LIN {X 0,Y 368.671,Z 450.598,A -85,B 0,C 180,E1 -13029.655,E2 -13029.655} C_VEL
LIN {X 0,Y 367.52,Z 522.522,A -85,B 0,C 180,E1 -13031.066,E2 -13031.066} C_VEL
LIN {X 0,Y 366.94,Z 535.872,A -85,B 0,C 180,E1 -13031.542,E2 -13031.542} C_VEL
LIN {X 0,Y 366.16,Z 548.093,A -85,B 0,C 180,E1 -13032.188,E2 -13032.188} C_VEL
LIN {X 0,Y 365.203,Z 560.412,A -85,B 0,C 180,E1 -13033.079,E2 -13033.079} C_VEL
LIN {X 0,Y 364.125,Z 572.06,A -85,B 0,C 180,E1 -13034.18,E2 -13034.18} C_VEL
LIN {X 0,Y 363.279,Z 582.567,A -85,B 0,C 180,E1 -13035.434,E2 -13035.434} C_VEL
LIN {X 0,Y 362.416,Z 591.99,A -85,B 0,C 180,E1 -13036.829,E2 -13036.829} C_VEL
LIN {X 0,Y 361.757,Z 599.735,A -85,B 0,C 180,E1 -13038.23,E2 -13038.23} C_VEL
LIN {X 0,Y 361.125,Z 607.312,A -85,B 0,C 180,E1 -13039.913,E2 -13039.913} C_VEL
LIN {X 0,Y 360.708,Z 613.396,A -85,B 0,C 180,E1 -13041.598,E2 -13041.598} C_VEL
LIN {X 0,Y 360.485,Z 618.204,A -85,B 0,C 180,E1 -13043.283,E2 -13043.283} C_VEL
LIN {X 0,Y 360.41,Z 621.877,A -85,B 0,C 180,E1 -13044.966,E2 -13044.966} C_VEL
LIN {X 0,Y 360.355,Z 624.517,A -85,B 0,C 180,E1 -13046.646,E2 -13046.646} C_VEL
LIN {X 0,Y 360.397,Z 625.759,A -85,B 0,C 180,E1 -13047.765,E2 -13047.765} C_VEL
LIN {X 0,Y 360.475,Z 626.58,A -85,B 0,C 180,E1 -13048.883,E2 -13048.883} C_VEL
LIN {X 0,Y 360.477,Z 626.968,A -85,B 0,C 180,E1 -13050,E2 -13050} C_VEL
LIN {X 0,Y 360.453,Z 626.966,A -85,B 0,C 180,E1 -13051.117,E2 -13051.117} C_VEL
LIN {X 0,Y 360.353,Z 626.574,A -85,B 0,C 180,E1 -13052.235,E2 -13052.235} C_VEL
LIN {X 0,Y 360.326,Z 625.784,A -85,B 0,C 180,E1 -13053.354,E2 -13053.354} C_VEL
LIN {X 0,Y 360.371,Z 624.558,A -85,B 0,C 180,E1 -13054.474,E2 -13054.474} C_VEL
LIN {X 0,Y 360.378,Z 622.329,A -85,B 0,C 180,E1 -13055.962,E2 -13055.962} C_VEL
LIN {X 0,Y 360.659,Z 618.37,A -85,B 0,C 180,E1 -13057.84,E2 -13057.84} C_VEL
LIN {X 0,Y 361.044,Z 613.682,A -85,B 0,C 180,E1 -13059.524,E2 -13059.524} C_VEL
LIN {X 0,Y 361.799,Z 606.644,A -85,B 0,C 180,E1 -13061.485,E2 -13061.485} C_VEL
LIN {X 0,Y 362.838,Z 599.055,A -85,B 0,C 180,E1 -13063.155,E2 -13063.155} C_VEL
LIN {X 0,Y 363.751,Z 591.32,A -85,B 0,C 180,E1 -13064.547,E2 -13064.547} C_VEL
LIN {X 0,Y 364.891,Z 581.912,A -85,B 0,C 180,E1 -13065.93,E2 -13065.93} C_VEL
LIN {X 0,Y 366.159,Z 571.498,A -85,B 0,C 180,E1 -13067.163,E2 -13067.163} C_VEL
LIN {X 0,Y 367.506,Z 559.948,A -85,B 0,C 180,E1 -13068.249,E2 -13068.249} C_VEL
LIN {X 0,Y 368.692,Z 547.75,A -85,B 0,C 180,E1 -13069.124,E2 -13069.124} C_VEL
LIN {X 0,Y 369.773,Z 534.193,A -85,B 0,C 180,E1 -13069.824,E2 -13069.824} C_VEL
LIN {X 0,Y 370.417,Z 521.877,A -85,B 0,C 180,E1 -13070.248,E2 -13070.248} C_VEL
LIN {X 0,Y 371.759,Z 449.686,A -85,B 0,C 180,E1 -13071.68,E2 -13071.68} C_VEL
LIN {X 0,Y 368.14,Z 427.447,A -85,B 0,C 180,E1 -13072.406,E2 -13072.406} C_VEL
LIN {X 0,Y 365.405,Z 413.474,A -85,B 0,C 180,E1 -13072.911,E2 -13072.911} C_VEL
LIN {X 0,Y 366.879,Z 400.729,A -85,B 0,C 180,E1 -13075.797,E2 -13075.797} C_VEL
LIN {X 0,Y 366.457,Z 396.694,A -85,B 0,C 180,E1 -13076.787,E2 -13076.787} C_VEL
LIN {X 0,Y 364.259,Z 386.406,A -85,B 0,C 180,E1 -13079.468,E2 -13079.468} C_VEL
LIN {X 0,Y 361.866,Z 376.41,A -85,B 0,C 180,E1 -13082.24,E2 -13082.24} C_VEL
LIN {X 0,Y 361.866,Z 376.411,A -85,B 0,C 180,E1 -13085.636,E2 -13085.636} C_VEL
LIN {X 0,Y 361.868,Z 376.407,A -85,B 0,C 180,E1 -13089.026,E2 -13089.026} C_VEL
LIN {X 0,Y 361.834,Z 376.409,A -85,B 0,C 180,E1 -13092.828,E2 -13092.828} C_VEL
LIN {X 0,Y 361.908,Z 376.401,A -85,B 0,C 180,E1 -13095.931,E2 -13095.931} C_VEL
LIN {X 0,Y 361.902,Z 376.401,A -85,B 0,C 180,E1 -13099.231,E2 -13099.231} C_VEL
LIN {X 0,Y 361.864,Z 376.405,A -85,B 0,C 180,E1 -13102.982,E2 -13102.982} C_VEL
LIN {X 0,Y 361.853,Z 376.408,A -85,B 0,C 180,E1 -13106.63,E2 -13106.63} C_VEL
LIN {X 0,Y 361.87,Z 376.406,A -85,B 0,C 180,E1 -13109.672,E2 -13109.672} C_VEL
LIN {X 0,Y 361.948,Z 376.387,A -85,B 0,C 180,E1 -13113.475,E2 -13113.475} C_VEL
LIN {X 0,Y 361.883,Z 376.399,A -85,B 0,C 180,E1 -13117.144,E2 -13117.144} C_VEL
LIN {X 0,Y 361.913,Z 376.398,A -85,B 0,C 180,E1 -13120.724,E2 -13120.724} C_VEL
LIN {X 0,Y 361.938,Z 376.395,A -85,B 0,C 180,E1 -13124.226,E2 -13124.226} C_VEL
LIN {X 0,Y 361.992,Z 376.391,A -85,B 0,C 180,E1 -13126.528,E2 -13126.528} C_VEL
LIN {X 0,Y 362.029,Z 376.382,A -85,B 0,C 180,E1 -13129.938,E2 -13129.938} C_VEL
LIN {X 0,Y 362.143,Z 376.373,A -85,B 0,C 180,E1 -13132.193,E2 -13132.193} C_VEL
LIN {X 0,Y 362.111,Z 376.37,A -85,B 0,C 180,E1 -13134.431,E2 -13134.431} C_VEL
LIN {X 0,Y 362.276,Z 376.353,A -85,B 0,C 180,E1 -13137.777,E2 -13137.777} C_VEL
LIN {X 0,Y 362.422,Z 376.336,A -85,B 0,C 180,E1 -13140,E2 -13140} C_VEL
LIN {X 0,Y 362.275,Z 376.357,A -85,B 0,C 180,E1 -13142.224,E2 -13142.224} C_VEL
LIN {X 0,Y 362.157,Z 376.373,A -85,B 0,C 180,E1 -13146.687,E2 -13146.687} C_VEL
LIN {X 0,Y 362.024,Z 376.388,A -85,B 0,C 180,E1 -13150.063,E2 -13150.063} C_VEL
LIN {X 0,Y 361.991,Z 376.39,A -85,B 0,C 180,E1 -13153.899,E2 -13153.899} C_VEL
LIN {X 0,Y 361.961,Z 376.393,A -85,B 0,C 180,E1 -13157.939,E2 -13157.939} C_VEL
LIN {X 0,Y 361.886,Z 376.402,A -85,B 0,C 180,E1 -13161.654,E2 -13161.654} C_VEL
LIN {X 0,Y 361.923,Z 376.39,A -85,B 0,C 180,E1 -13165.291,E2 -13165.291} C_VEL
LIN {X 0,Y 361.913,Z 376.391,A -85,B 0,C 180,E1 -13167.779,E2 -13167.779} C_VEL
LIN {X 0,Y 361.842,Z 376.407,A -85,B 0,C 180,E1 -13171.286,E2 -13171.286} C_VEL
LIN {X 0,Y 361.85,Z 376.411,A -85,B 0,C 180,E1 -13174.281,E2 -13174.281} C_VEL
LIN {X 0,Y 361.862,Z 376.408,A -85,B 0,C 180,E1 -13177.224,E2 -13177.224} C_VEL
LIN {X 0,Y 361.903,Z 376.407,A -85,B 0,C 180,E1 -13180.769,E2 -13180.769} C_VEL
LIN {X 0,Y 361.909,Z 376.411,A -85,B 0,C 180,E1 -13184.355,E2 -13184.355} C_VEL
LIN {X 0,Y 361.857,Z 376.415,A -85,B 0,C 180,E1 -13187.565,E2 -13187.565} C_VEL
LIN {X 0,Y 361.875,Z 376.41,A -85,B 0,C 180,E1 -13190.973,E2 -13190.973} C_VEL
LIN {X 0,Y 361.875,Z 376.41,A -85,B 0,C 180,E1 -13194.656,E2 -13194.656} C_VEL
LIN {X 0,Y 361.934,Z 376.564,A -85,B 0,C 180,E1 -13195.729,E2 -13195.729} C_VEL
LIN {X 0,Y 363.517,Z 383.858,A -85,B 0,C 180,E1 -13198.004,E2 -13198.004} C_VEL
LIN {X 0,Y 370.823,Z 401.263,A -85,B 0,C 180,E1 -13198.929,E2 -13198.929} C_VEL
LIN {X 0,Y 372.558,Z 408.259,A -85,B 0,C 180,E1 -13199.203,E2 -13199.203} C_VEL
LIN {X 0,Y 370.891,Z 490.155,A -85,B 0,C 180,E1 -13200.824,E2 -13200.824} C_VEL
LIN {X 0,Y 370.371,Z 502.076,A -85,B 0,C 180,E1 -13201.247,E2 -13201.247} C_VEL
LIN {X 0,Y 369.552,Z 514.899,A -85,B 0,C 180,E1 -13201.922,E2 -13201.922} C_VEL
LIN {X 0,Y 368.697,Z 524.869,A -85,B 0,C 180,E1 -13202.622,E2 -13202.622} C_VEL
LIN {X 0,Y 367.786,Z 535.953,A -85,B 0,C 180,E1 -13203.623,E2 -13203.623} C_VEL
LIN {X 0,Y 366.561,Z 546.433,A -85,B 0,C 180,E1 -13204.805,E2 -13204.805} C_VEL
LIN {X 0,Y 365.343,Z 556.155,A -85,B 0,C 180,E1 -13206.174,E2 -13206.174} C_VEL
LIN {X 0,Y 364.217,Z 564.926,A -85,B 0,C 180,E1 -13207.702,E2 -13207.702} C_VEL
LIN {X 0,Y 363.166,Z 572.436,A -85,B 0,C 180,E1 -13209.319,E2 -13209.319} C_VEL
LIN {X 0,Y 362.381,Z 577.833,A -85,B 0,C 180,E1 -13210.75,E2 -13210.75} C_VEL
LIN {X 0,Y 361.675,Z 583.349,A -85,B 0,C 180,E1 -13212.581,E2 -13212.581} C_VEL
LIN {X 0,Y 361.165,Z 587.097,A -85,B 0,C 180,E1 -13214.192,E2 -13214.192} C_VEL
LIN {X 0,Y 360.907,Z 589.153,A -85,B 0,C 180,E1 -13215.336,E2 -13215.336} C_VEL
LIN {X 0,Y 360.684,Z 591.358,A -85,B 0,C 180,E1 -13216.975,E2 -13216.975} C_VEL
LIN {X 0,Y 360.421,Z 592.768,A -85,B 0,C 180,E1 -13218.756,E2 -13218.756} C_VEL
LIN {X 0,Y 360.326,Z 593.102,A -85,B 0,C 180,E1 -13221.023,E2 -13221.023} C_VEL
LIN {X 0,Y 360.391,Z 592.689,A -85,B 0,C 180,E1 -13222.154,E2 -13222.154} C_VEL
LIN {X 0,Y 360.52,Z 591.294,A -85,B 0,C 180,E1 -13223.83,E2 -13223.83} C_VEL
LIN {X 0,Y 360.617,Z 587.969,A -85,B 0,C 180,E1 -13226.089,E2 -13226.089} C_VEL
LIN {X 0,Y 360.94,Z 584.326,A -85,B 0,C 180,E1 -13227.768,E2 -13227.768} C_VEL
LIN {X 0,Y 361.199,Z 579.599,A -85,B 0,C 180,E1 -13229.443,E2 -13229.443} C_VEL
LIN {X 0,Y 361.97,Z 572.495,A -85,B 0,C 180,E1 -13231.391,E2 -13231.391} C_VEL
LIN {X 0,Y 362.707,Z 564.761,A -85,B 0,C 180,E1 -13233.054,E2 -13233.054} C_VEL
LIN {X 0,Y 363.587,Z 555.113,A -85,B 0,C 180,E1 -13234.712,E2 -13234.712} C_VEL
LIN {X 0,Y 364.548,Z 545.11,A -85,B 0,C 180,E1 -13236.087,E2 -13236.087} C_VEL
LIN {X 0,Y 365.502,Z 533.787,A -85,B 0,C 180,E1 -13237.319,E2 -13237.319} C_VEL
LIN {X 0,Y 366.31,Z 522.692,A -85,B 0,C 180,E1 -13238.273,E2 -13238.273} C_VEL
LIN {X 0,Y 366.903,Z 511.497,A -85,B 0,C 180,E1 -13239.023,E2 -13239.023} C_VEL
LIN {X 0,Y 367.47,Z 498.848,A -85,B 0,C 180,E1 -13239.633,E2 -13239.633} C_VEL
LIN {X 0,Y 367.834,Z 485.603,A -85,B 0,C 180,E1 -13240.039,E2 -13240.039} C_VEL
LIN {X 0,Y 369.128,Z 406.287,A -85,B 0,C 180,E1 -13241.575,E2 -13241.575} C_VEL
LIN {X 0,Y 367.573,Z 397.862,A -85,B 0,C 180,E1 -13241.824,E2 -13241.824} C_VEL
LIN {X 0,Y 366.097,Z 394.053,A -85,B 0,C 180,E1 -13241.983,E2 -13241.983} C_VEL
LIN {X 0,Y 363.787,Z 390.703,A -85,B 0,C 180,E1 -13242.176,E2 -13242.176} C_VEL
LIN {X 0,Y 357.343,Z 384.3,A -85,B 0,C 180,E1 -13242.689,E2 -13242.689} C_VEL
LIN {X 0,Y 355.96,Z 382.402,A -85,B 0,C 180,E1 -13243.038,E2 -13243.038} C_VEL
LIN {X 0,Y 355.86,Z 382.081,A -85,B 0,C 180,E1 -13243.125,E2 -13243.125} C_VEL
LIN {X 0,Y 354.939,Z 377.274,A -85,B 0,C 180,E1 -13244.616,E2 -13244.616} C_VEL
LIN {X 0,Y 354.911,Z 377.279,A -85,B 0,C 180,E1 -13248.471,E2 -13248.471} C_VEL
LIN {X 0,Y 354.839,Z 377.284,A -85,B 0,C 180,E1 -13252.105,E2 -13252.105} C_VEL
LIN {X 0,Y 354.902,Z 377.274,A -85,B 0,C 180,E1 -13255.827,E2 -13255.827} C_VEL
LIN {X 0,Y 354.856,Z 377.279,A -85,B 0,C 180,E1 -13259.678,E2 -13259.678} C_VEL
LIN {X 0,Y 354.807,Z 377.286,A -85,B 0,C 180,E1 -13263.701,E2 -13263.701} C_VEL
LIN {X 0,Y 354.8,Z 377.292,A -85,B 0,C 180,E1 -13266.458,E2 -13266.458} C_VEL
LIN {X 0,Y 354.824,Z 377.283,A -85,B 0,C 180,E1 -13269.423,E2 -13269.423} C_VEL
LIN {X 0,Y 354.789,Z 377.289,A -85,B 0,C 180,E1 -13272.867,E2 -13272.867} C_VEL
LIN {X 0,Y 354.851,Z 377.284,A -85,B 0,C 180,E1 -13276.116,E2 -13276.116} C_VEL
LIN {X 0,Y 354.854,Z 377.279,A -85,B 0,C 180,E1 -13279.188,E2 -13279.188} C_VEL
LIN {X 0,Y 354.81,Z 377.29,A -85,B 0,C 180,E1 -13282.4,E2 -13282.4} C_VEL
LIN {X 0,Y 354.808,Z 377.286,A -85,B 0,C 180,E1 -13284.94,E2 -13284.94} C_VEL
LIN {X 0,Y 354.789,Z 377.292,A -85,B 0,C 180,E1 -13288.404,E2 -13288.404} C_VEL
LIN {X 0,Y 354.841,Z 377.282,A -85,B 0,C 180,E1 -13291.618,E2 -13291.618} C_VEL
LIN {X 0,Y 354.894,Z 377.28,A -85,B 0,C 180,E1 -13294.172,E2 -13294.172} C_VEL
LIN {X 0,Y 354.835,Z 377.285,A -85,B 0,C 180,E1 -13297.894,E2 -13297.894} C_VEL
LIN {X 0,Y 354.917,Z 377.275,A -85,B 0,C 180,E1 -13301.89,E2 -13301.89} C_VEL
LIN {X 0,Y 354.936,Z 377.273,A -85,B 0,C 180,E1 -13305.98,E2 -13305.98} C_VEL
LIN {X 0,Y 354.976,Z 377.266,A -85,B 0,C 180,E1 -13309.735,E2 -13309.735} C_VEL
LIN {X 0,Y 355.107,Z 377.253,A -85,B 0,C 180,E1 -13312.036,E2 -13312.036} C_VEL
LIN {X 0,Y 355.085,Z 377.255,A -85,B 0,C 180,E1 -13314.32,E2 -13314.32} C_VEL
LIN {X 0,Y 355.239,Z 377.234,A -85,B 0,C 180,E1 -13317.732,E2 -13317.732} C_VEL
LIN {X 0,Y 355.391,Z 377.218,A -85,B 0,C 180,E1 -13320,E2 -13320} C_VEL
LIN {X 0,Y 355.239,Z 377.236,A -85,B 0,C 180,E1 -13322.267,E2 -13322.267} C_VEL
LIN {X 0,Y 355.13,Z 377.245,A -85,B 0,C 180,E1 -13326.819,E2 -13326.819} C_VEL
LIN {X 0,Y 355.009,Z 377.26,A -85,B 0,C 180,E1 -13329.112,E2 -13329.112} C_VEL
LIN {X 0,Y 354.919,Z 377.273,A -85,B 0,C 180,E1 -13332.581,E2 -13332.581} C_VEL
LIN {X 0,Y 354.883,Z 377.282,A -85,B 0,C 180,E1 -13336.096,E2 -13336.096} C_VEL
LIN {X 0,Y 354.901,Z 377.275,A -85,B 0,C 180,E1 -13338.472,E2 -13338.472} C_VEL
LIN {X 0,Y 354.834,Z 377.287,A -85,B 0,C 180,E1 -13342.106,E2 -13342.106} C_VEL
LIN {X 0,Y 354.892,Z 377.279,A -85,B 0,C 180,E1 -13345.828,E2 -13345.828} C_VEL
LIN {X 0,Y 354.811,Z 377.288,A -85,B 0,C 180,E1 -13349.682,E2 -13349.682} C_VEL
LIN {X 0,Y 354.8,Z 377.29,A -85,B 0,C 180,E1 -13353.703,E2 -13353.703} C_VEL
LIN {X 0,Y 354.794,Z 377.288,A -85,B 0,C 180,E1 -13356.46,E2 -13356.46} C_VEL
LIN {X 0,Y 354.819,Z 377.285,A -85,B 0,C 180,E1 -13359.424,E2 -13359.424} C_VEL
LIN {X 0,Y 354.831,Z 377.282,A -85,B 0,C 180,E1 -13362.876,E2 -13362.876} C_VEL
LIN {X 0,Y 354.793,Z 377.291,A -85,B 0,C 180,E1 -13366.109,E2 -13366.109} C_VEL
LIN {X 0,Y 354.784,Z 377.289,A -85,B 0,C 180,E1 -13369.18,E2 -13369.18} C_VEL
LIN {X 0,Y 354.805,Z 377.287,A -85,B 0,C 180,E1 -13372.403,E2 -13372.403} C_VEL
LIN {X 0,Y 354.81,Z 377.285,A -85,B 0,C 180,E1 -13374.942,E2 -13374.942} C_VEL
LIN {X 0,Y 354.815,Z 377.285,A -85,B 0,C 180,E1 -13378.4,E2 -13378.4} C_VEL
LIN {X 0,Y 354.915,Z 377.465,A -85,B 0,C 180,E1 -13379.755,E2 -13379.755} C_VEL
LIN {X 0,Y 357.366,Z 389.378,A -85,B 0,C 180,E1 -13382.743,E2 -13382.743} C_VEL
LIN {X 0,Y 358.518,Z 396.453,A -85,B 0,C 180,E1 -13384.453,E2 -13384.453} C_VEL
LIN {X 0,Y 357.181,Z 410.658,A -85,B 0,C 180,E1 -13387.636,E2 -13387.636} C_VEL
LIN {X 0,Y 356.914,Z 413.639,A -85,B 0,C 180,E1 -13388.301,E2 -13388.301} C_VEL
LIN {X 0,Y 361.882,Z 450.204,A -85,B 0,C 180,E1 -13389.317,E2 -13389.317} C_VEL
LIN {X 0,Y 360.697,Z 522.605,A -85,B 0,C 180,E1 -13390.768,E2 -13390.768} C_VEL
LIN {X 0,Y 360.091,Z 535.816,A -85,B 0,C 180,E1 -13391.251,E2 -13391.251} C_VEL
LIN {X 0,Y 359.286,Z 547.966,A -85,B 0,C 180,E1 -13391.909,E2 -13391.909} C_VEL
LIN {X 0,Y 358.41,Z 559.427,A -85,B 0,C 180,E1 -13392.748,E2 -13392.748} C_VEL
LIN {X 0,Y 357.294,Z 571.201,A -85,B 0,C 180,E1 -13393.869,E2 -13393.869} C_VEL
LIN {X 0,Y 356.305,Z 581.79,A -85,B 0,C 180,E1 -13395.143,E2 -13395.143} C_VEL
LIN {X 0,Y 355.46,Z 591.324,A -85,B 0,C 180,E1 -13396.567,E2 -13396.567} C_VEL
LIN {X 0,Y 354.766,Z 599.127,A -85,B 0,C 180,E1 -13397.995,E2 -13397.995} C_VEL
LIN {X 0,Y 354.077,Z 606.751,A -85,B 0,C 180,E1 -13399.71,E2 -13399.71} C_VEL
LIN {X 0,Y 353.652,Z 612.881,A -85,B 0,C 180,E1 -13401.429,E2 -13401.429} C_VEL
LIN {X 0,Y 353.396,Z 617.727,A -85,B 0,C 180,E1 -13403.147,E2 -13403.147} C_VEL
LIN {X 0,Y 353.31,Z 621.436,A -85,B 0,C 180,E1 -13404.865,E2 -13404.865} C_VEL
LIN {X 0,Y 353.274,Z 624.111,A -85,B 0,C 180,E1 -13406.579,E2 -13406.579} C_VEL
LIN {X 0,Y 353.3,Z 625.37,A -85,B 0,C 180,E1 -13407.72,E2 -13407.72} C_VEL
LIN {X 0,Y 353.393,Z 626.221,A -85,B 0,C 180,E1 -13408.86,E2 -13408.86} C_VEL
LIN {X 0,Y 353.395,Z 626.626,A -85,B 0,C 180,E1 -13410,E2 -13410} C_VEL
LIN {X 0,Y 353.355,Z 626.639,A -85,B 0,C 180,E1 -13411.14,E2 -13411.14} C_VEL
LIN {X 0,Y 353.245,Z 625.498,A -85,B 0,C 180,E1 -13413.422,E2 -13413.422} C_VEL
LIN {X 0,Y 353.282,Z 624.294,A -85,B 0,C 180,E1 -13414.564,E2 -13414.564} C_VEL
LIN {X 0,Y 353.414,Z 620.653,A -85,B 0,C 180,E1 -13416.852,E2 -13416.852} C_VEL
LIN {X 0,Y 353.718,Z 616.737,A -85,B 0,C 180,E1 -13418.57,E2 -13418.57} C_VEL
LIN {X 0,Y 354.223,Z 611.706,A -85,B 0,C 180,E1 -13420.286,E2 -13420.286} C_VEL
LIN {X 0,Y 354.96,Z 605.411,A -85,B 0,C 180,E1 -13421.999,E2 -13421.999} C_VEL
LIN {X 0,Y 356.115,Z 597.563,A -85,B 0,C 180,E1 -13423.699,E2 -13423.699} C_VEL
LIN {X 0,Y 357.115,Z 589.198,A -85,B 0,C 180,E1 -13425.178,E2 -13425.178} C_VEL
LIN {X 0,Y 358.438,Z 578.813,A -85,B 0,C 180,E1 -13426.663,E2 -13426.663} C_VEL
LIN {X 0,Y 359.918,Z 567.735,A -85,B 0,C 180,E1 -13427.911,E2 -13427.911} C_VEL
LIN {X 0,Y 361.157,Z 556.909,A -85,B 0,C 180,E1 -13428.875,E2 -13428.875} C_VEL
LIN {X 0,Y 362.339,Z 544.985,A -85,B 0,C 180,E1 -13429.694,E2 -13429.694} C_VEL
LIN {X 0,Y 363.37,Z 532.038,A -85,B 0,C 180,E1 -13430.336,E2 -13430.336} C_VEL
LIN {X 0,Y 363.954,Z 519.458,A -85,B 0,C 180,E1 -13430.74,E2 -13430.74} C_VEL
LIN {X 0,Y 365.32,Z 450.584,A -85,B 0,C 180,E1 -13432.12,E2 -13432.12} C_VEL
LIN {X 0,Y 361.717,Z 428.652,A -85,B 0,C 180,E1 -13432.857,E2 -13432.857} C_VEL
LIN {X 0,Y 358.692,Z 413.022,A -85,B 0,C 180,E1 -13433.461,E2 -13433.461} C_VEL
LIN {X 0,Y 360.023,Z 401.589,A -85,B 0,C 180,E1 -13436.108,E2 -13436.108} C_VEL
LIN {X 0,Y 358.696,Z 393.663,A -85,B 0,C 180,E1 -13438.153,E2 -13438.153} C_VEL
LIN {X 0,Y 355.79,Z 381.304,A -85,B 0,C 180,E1 -13441.556,E2 -13441.556} C_VEL
LIN {X 0,Y 354.814,Z 377.288,A -85,B 0,C 180,E1 -13442.75,E2 -13442.75} C_VEL
LIN {X 0,Y 354.797,Z 377.291,A -85,B 0,C 180,E1 -13446.459,E2 -13446.459} C_VEL
LIN {X 0,Y 354.821,Z 377.287,A -85,B 0,C 180,E1 -13449.423,E2 -13449.423} C_VEL
LIN {X 0,Y 354.787,Z 377.287,A -85,B 0,C 180,E1 -13452.867,E2 -13452.867} C_VEL
LIN {X 0,Y 354.848,Z 377.28,A -85,B 0,C 180,E1 -13456.116,E2 -13456.116} C_VEL
LIN {X 0,Y 354.853,Z 377.278,A -85,B 0,C 180,E1 -13459.188,E2 -13459.188} C_VEL
LIN {X 0,Y 354.804,Z 377.284,A -85,B 0,C 180,E1 -13462.402,E2 -13462.402} C_VEL
LIN {X 0,Y 354.807,Z 377.286,A -85,B 0,C 180,E1 -13464.94,E2 -13464.94} C_VEL
LIN {X 0,Y 354.787,Z 377.289,A -85,B 0,C 180,E1 -13468.405,E2 -13468.405} C_VEL
LIN {X 0,Y 354.847,Z 377.285,A -85,B 0,C 180,E1 -13471.619,E2 -13471.619} C_VEL
LIN {X 0,Y 354.893,Z 377.26,A -85,B 0,C 180,E1 -13474.172,E2 -13474.172} C_VEL
LIN {X 0,Y 354.828,Z 377.285,A -85,B 0,C 180,E1 -13477.894,E2 -13477.894} C_VEL
LIN {X 0,Y 354.916,Z 377.273,A -85,B 0,C 180,E1 -13481.891,E2 -13481.891} C_VEL
LIN {X 0,Y 354.936,Z 377.269,A -85,B 0,C 180,E1 -13485.981,E2 -13485.981} C_VEL
LIN {X 0,Y 354.975,Z 377.262,A -85,B 0,C 180,E1 -13489.736,E2 -13489.736} C_VEL
LIN {X 0,Y 355.106,Z 377.249,A -85,B 0,C 180,E1 -13492.037,E2 -13492.037} C_VEL
LIN {X 0,Y 355.085,Z 377.245,A -85,B 0,C 180,E1 -13494.321,E2 -13494.321} C_VEL
LIN {X 0,Y 355.239,Z 377.23,A -85,B 0,C 180,E1 -13497.733,E2 -13497.733} C_VEL
LIN {X 0,Y 355.391,Z 377.211,A -85,B 0,C 180,E1 -13500,E2 -13500} C_VEL
LIN {X 0,Y 355.239,Z 377.234,A -85,B 0,C 180,E1 -13502.268,E2 -13502.268} C_VEL
LIN {X 0,Y 355.12,Z 377.248,A -85,B 0,C 180,E1 -13506.82,E2 -13506.82} C_VEL
LIN {X 0,Y 354.971,Z 377.268,A -85,B 0,C 180,E1 -13510.265,E2 -13510.265} C_VEL
LIN {X 0,Y 354.936,Z 377.269,A -85,B 0,C 180,E1 -13514.019,E2 -13514.019} C_VEL
LIN {X 0,Y 354.917,Z 377.272,A -85,B 0,C 180,E1 -13518.109,E2 -13518.109} C_VEL
LIN {X 0,Y 354.829,Z 377.283,A -85,B 0,C 180,E1 -13522.107,E2 -13522.107} C_VEL
LIN {X 0,Y 354.894,Z 377.26,A -85,B 0,C 180,E1 -13525.828,E2 -13525.828} C_VEL
LIN {X 0,Y 354.849,Z 377.283,A -85,B 0,C 180,E1 -13529.68,E2 -13529.68} C_VEL
LIN {X 0,Y 354.802,Z 377.289,A -85,B 0,C 180,E1 -13533.703,E2 -13533.703} C_VEL
LIN {X 0,Y 354.796,Z 377.289,A -85,B 0,C 180,E1 -13536.46,E2 -13536.46} C_VEL
LIN {X 0,Y 354.821,Z 377.286,A -85,B 0,C 180,E1 -13539.425,E2 -13539.425} C_VEL
LIN {X 0,Y 354.833,Z 377.281,A -85,B 0,C 180,E1 -13542.876,E2 -13542.876} C_VEL
LIN {X 0,Y 354.803,Z 377.288,A -85,B 0,C 180,E1 -13546.11,E2 -13546.11} C_VEL
LIN {X 0,Y 354.824,Z 377.291,A -85,B 0,C 180,E1 -13549.185,E2 -13549.185} C_VEL
LIN {X 0,Y 354.814,Z 377.29,A -85,B 0,C 180,E1 -13552.402,E2 -13552.402} C_VEL
LIN {X 0,Y 354.885,Z 377.453,A -85,B 0,C 180,E1 -13555.279,E2 -13555.279} C_VEL
LIN {X 0,Y 356.325,Z 384.015,A -85,B 0,C 180,E1 -13557.43,E2 -13557.43} C_VEL
LIN {X 0,Y 364.572,Z 403.454,A -85,B 0,C 180,E1 -13558.508,E2 -13558.508} C_VEL
LIN {X 0,Y 366.143,Z 409.637,A -85,B 0,C 180,E1 -13558.759,E2 -13558.759} C_VEL
LIN {X 0,Y 364.405,Z 490.429,A -85,B 0,C 180,E1 -13560.384,E2 -13560.384} C_VEL
LIN {X 0,Y 363.844,Z 502.682,A -85,B 0,C 180,E1 -13560.828,E2 -13560.828} C_VEL
LIN {X 0,Y 362.97,Z 515.611,A -85,B 0,C 180,E1 -13561.524,E2 -13561.524} C_VEL
LIN {X 0,Y 361.93,Z 527.283,A -85,B 0,C 180,E1 -13562.381,E2 -13562.381} C_VEL
LIN {X 0,Y 360.808,Z 539.191,A -85,B 0,C 180,E1 -13563.54,E2 -13563.54} C_VEL
LIN {X 0,Y 359.482,Z 549.814,A -85,B 0,C 180,E1 -13564.836,E2 -13564.836} C_VEL
LIN {X 0,Y 358.217,Z 559.29,A -85,B 0,C 180,E1 -13566.285,E2 -13566.285} C_VEL
LIN {X 0,Y 356.967,Z 568.401,A -85,B 0,C 180,E1 -13568.033,E2 -13568.033} C_VEL
LIN {X 0,Y 355.835,Z 575.683,A -85,B 0,C 180,E1 -13569.78,E2 -13569.78} C_VEL
LIN {X 0,Y 354.992,Z 581.435,A -85,B 0,C 180,E1 -13571.533,E2 -13571.533} C_VEL
LIN {X 0,Y 354.39,Z 585.924,A -85,B 0,C 180,E1 -13573.289,E2 -13573.289} C_VEL
LIN {X 0,Y 353.902,Z 589.298,A -85,B 0,C 180,E1 -13575.039,E2 -13575.039} C_VEL
LIN {X 0,Y 353.605,Z 591.738,A -85,B 0,C 180,E1 -13576.881,E2 -13576.881} C_VEL
LIN {X 0,Y 353.377,Z 593.049,A -85,B 0,C 180,E1 -13578.529,E2 -13578.529} C_VEL
LIN {X 0,Y 353.225,Z 593.456,A -85,B 0,C 180,E1 -13580.841,E2 -13580.841} C_VEL
LIN {X 0,Y 353.292,Z 593.077,A -85,B 0,C 180,E1 -13581.996,E2 -13581.996} C_VEL
LIN {X 0,Y 353.428,Z 591.593,A -85,B 0,C 180,E1 -13583.865,E2 -13583.865} C_VEL
LIN {X 0,Y 353.525,Z 588.529,A -85,B 0,C 180,E1 -13586.01,E2 -13586.01} C_VEL
LIN {X 0,Y 353.86,Z 584.962,A -85,B 0,C 180,E1 -13587.724,E2 -13587.724} C_VEL
LIN {X 0,Y 354.118,Z 580.315,A -85,B 0,C 180,E1 -13589.431,E2 -13589.431} C_VEL
LIN {X 0,Y 354.875,Z 573.303,A -85,B 0,C 180,E1 -13591.418,E2 -13591.418} C_VEL
LIN {X 0,Y 355.663,Z 565.716,A -85,B 0,C 180,E1 -13593.115,E2 -13593.115} C_VEL
LIN {X 0,Y 356.545,Z 556.199,A -85,B 0,C 180,E1 -13594.805,E2 -13594.805} C_VEL
LIN {X 0,Y 357.558,Z 546.368,A -85,B 0,C 180,E1 -13596.206,E2 -13596.206} C_VEL
LIN {X 0,Y 358.527,Z 535.319,A -85,B 0,C 180,E1 -13597.462,E2 -13597.462} C_VEL
LIN {X 0,Y 359.464,Z 522.764,A -85,B 0,C 180,E1 -13598.573,E2 -13598.573} C_VEL
LIN {X 0,Y 360.103,Z 511.482,A -85,B 0,C 180,E1 -13599.336,E2 -13599.336} C_VEL
LIN {X 0,Y 360.681,Z 498.629,A -85,B 0,C 180,E1 -13599.958,E2 -13599.958} C_VEL
LIN {X 0,Y 361.044,Z 484.988,A -85,B 0,C 180,E1 -13600.373,E2 -13600.373} C_VEL
LIN {X 0,Y 362.284,Z 406.824,A -85,B 0,C 180,E1 -13601.915,E2 -13601.915} C_VEL
LIN {X 0,Y 359.867,Z 394.984,A -85,B 0,C 180,E1 -13602.287,E2 -13602.287} C_VEL
LIN {X 0,Y 356.128,Z 383.323,A -85,B 0,C 180,E1 -13602.754,E2 -13602.754} C_VEL
LIN {X 0,Y 355.86,Z 382.081,A -85,B 0,C 180,E1 -13603.125,E2 -13603.125} C_VEL
LIN {X 0,Y 354.851,Z 380.454,A -85,B 0,C 180,E1 -13603.693,E2 -13603.693} C_VEL
LIN {X 0,Y 353.008,Z 379.35,A -85,B 0,C 180,E1 -13604.253,E2 -13604.253} C_VEL
LIN {X 0,Y 349.026,Z 378.306,A -85,B 0,C 180,E1 -13605.411,E2 -13605.411} C_VEL
LIN {X 0,Y 347.86,Z 378.16,A -85,B 0,C 180,E1 -13606.159,E2 -13606.159} C_VEL
LIN {X 0,Y 347.84,Z 378.158,A -85,B 0,C 180,E1 -13606.269,E2 -13606.269} C_VEL
LIN {X 0,Y 347.86,Z 378.153,A -85,B 0,C 180,E1 -13608.86,E2 -13608.86} C_VEL
LIN {X 0,Y 347.778,Z 378.166,A -85,B 0,C 180,E1 -13612.578,E2 -13612.578} C_VEL
LIN {X 0,Y 347.815,Z 378.156,A -85,B 0,C 180,E1 -13615.108,E2 -13615.108} C_VEL
LIN {X 0,Y 347.815,Z 378.157,A -85,B 0,C 180,E1 -13617.693,E2 -13617.693} C_VEL
LIN {X 0,Y 347.766,Z 378.168,A -85,B 0,C 180,E1 -13620.345,E2 -13620.345} C_VEL
LIN {X 0,Y 347.745,Z 378.17,A -85,B 0,C 180,E1 -13624.463,E2 -13624.463} C_VEL
LIN {X 0,Y 347.774,Z 378.164,A -85,B 0,C 180,E1 -13627.988,E2 -13627.988} C_VEL
LIN {X 0,Y 347.75,Z 378.165,A -85,B 0,C 180,E1 -13631.829,E2 -13631.829} C_VEL
LIN {X 0,Y 347.797,Z 378.159,A -85,B 0,C 180,E1 -13635.01,E2 -13635.01} C_VEL
LIN {X 0,Y 347.782,Z 378.166,A -85,B 0,C 180,E1 -13638.39,E2 -13638.39} C_VEL
LIN {X 0,Y 347.776,Z 378.164,A -85,B 0,C 180,E1 -13642.009,E2 -13642.009} C_VEL
LIN {X 0,Y 347.741,Z 378.165,A -85,B 0,C 180,E1 -13645.535,E2 -13645.535} C_VEL
LIN {X 0,Y 347.741,Z 378.171,A -85,B 0,C 180,E1 -13648.299,E2 -13648.299} C_VEL
LIN {X 0,Y 347.774,Z 378.162,A -85,B 0,C 180,E1 -13650.987,E2 -13650.987} C_VEL
LIN {X 0,Y 347.825,Z 378.155,A -85,B 0,C 180,E1 -13653.607,E2 -13653.607} C_VEL
LIN {X 0,Y 347.784,Z 378.165,A -85,B 0,C 180,E1 -13656.161,E2 -13656.161} C_VEL
LIN {X 0,Y 347.822,Z 378.158,A -85,B 0,C 180,E1 -13659.909,E2 -13659.909} C_VEL
LIN {X 0,Y 347.861,Z 378.155,A -85,B 0,C 180,E1 -13662.359,E2 -13662.359} C_VEL
LIN {X 0,Y 347.891,Z 378.15,A -85,B 0,C 180,E1 -13665.97,E2 -13665.97} C_VEL
LIN {X 0,Y 347.926,Z 378.143,A -85,B 0,C 180,E1 -13669.525,E2 -13669.525} C_VEL
LIN {X 0,Y 348.067,Z 378.128,A -85,B 0,C 180,E1 -13671.874,E2 -13671.874} C_VEL
LIN {X 0,Y 348.06,Z 378.131,A -85,B 0,C 180,E1 -13674.205,E2 -13674.205} C_VEL
LIN {X 0,Y 348.201,Z 378.11,A -85,B 0,C 180,E1 -13677.686,E2 -13677.686} C_VEL
LIN {X 0,Y 348.361,Z 378.093,A -85,B 0,C 180,E1 -13680,E2 -13680} C_VEL
LIN {X 0,Y 348.201,Z 378.112,A -85,B 0,C 180,E1 -13682.313,E2 -13682.313} C_VEL
LIN {X 0,Y 348.099,Z 378.121,A -85,B 0,C 180,E1 -13686.958,E2 -13686.958} C_VEL
LIN {X 0,Y 347.962,Z 378.138,A -85,B 0,C 180,E1 -13689.298,E2 -13689.298} C_VEL
LIN {X 0,Y 347.887,Z 378.147,A -85,B 0,C 180,E1 -13692.839,E2 -13692.839} C_VEL
LIN {X 0,Y 347.832,Z 378.156,A -85,B 0,C 180,E1 -13696.431,E2 -13696.431} C_VEL
LIN {X 0,Y 347.853,Z 378.151,A -85,B 0,C 180,E1 -13698.86,E2 -13698.86} C_VEL
LIN {X 0,Y 347.771,Z 378.163,A -85,B 0,C 180,E1 -13702.579,E2 -13702.579} C_VEL
LIN {X 0,Y 347.805,Z 378.157,A -85,B 0,C 180,E1 -13705.109,E2 -13705.109} C_VEL
LIN {X 0,Y 347.802,Z 378.161,A -85,B 0,C 180,E1 -13707.695,E2 -13707.695} C_VEL
LIN {X 0,Y 347.743,Z 378.168,A -85,B 0,C 180,E1 -13710.348,E2 -13710.348} C_VEL
LIN {X 0,Y 347.743,Z 378.17,A -85,B 0,C 180,E1 -13714.044,E2 -13714.044} C_VEL
LIN {X 0,Y 347.758,Z 378.164,A -85,B 0,C 180,E1 -13717.321,E2 -13717.321} C_VEL
LIN {X 0,Y 347.789,Z 378.162,A -85,B 0,C 180,E1 -13720.289,E2 -13720.289} C_VEL
LIN {X 0,Y 347.782,Z 378.162,A -85,B 0,C 180,E1 -13723.399,E2 -13723.399} C_VEL
LIN {X 0,Y 347.743,Z 378.165,A -85,B 0,C 180,E1 -13726.683,E2 -13726.683} C_VEL
LIN {X 0,Y 347.744,Z 378.168,A -85,B 0,C 180,E1 -13730.174,E2 -13730.174} C_VEL
LIN {X 0,Y 347.76,Z 378.163,A -85,B 0,C 180,E1 -13732.68,E2 -13732.68} C_VEL
LIN {X 0,Y 347.746,Z 378.17,A -85,B 0,C 180,E1 -13735.957,E2 -13735.957} C_VEL
LIN {X 0,Y 347.83,Z 378.182,A -85,B 0,C 180,E1 -13739.409,E2 -13739.409} C_VEL
LIN {X 0,Y 350.321,Z 390.288,A -85,B 0,C 180,E1 -13742.522,E2 -13742.522} C_VEL
LIN {X 0,Y 351.482,Z 396.784,A -85,B 0,C 180,E1 -13744.131,E2 -13744.131} C_VEL
LIN {X 0,Y 351.107,Z 402.527,A -85,B 0,C 180,E1 -13745.46,E2 -13745.46} C_VEL
LIN {X 0,Y 350.012,Z 413.325,A -85,B 0,C 180,E1 -13747.92,E2 -13747.92} C_VEL
LIN {X 0,Y 355.069,Z 450.43,A -85,B 0,C 180,E1 -13748.977,E2 -13748.977} C_VEL
LIN {X 0,Y 353.884,Z 522.633,A -85,B 0,C 180,E1 -13750.458,E2 -13750.458} C_VEL
LIN {X 0,Y 353.215,Z 536.495,A -85,B 0,C 180,E1 -13750.985,E2 -13750.985} C_VEL
LIN {X 0,Y 352.346,Z 548.914,A -85,B 0,C 180,E1 -13751.691,E2 -13751.691} C_VEL
LIN {X 0,Y 351.259,Z 561.62,A -85,B 0,C 180,E1 -13752.686,E2 -13752.686} C_VEL
LIN {X 0,Y 350.127,Z 572.929,A -85,B 0,C 180,E1 -13753.829,E2 -13753.829} C_VEL
LIN {X 0,Y 349.239,Z 583.463,A -85,B 0,C 180,E1 -13755.185,E2 -13755.185} C_VEL
LIN {X 0,Y 348.335,Z 592.302,A -85,B 0,C 180,E1 -13756.584,E2 -13756.584} C_VEL
LIN {X 0,Y 347.471,Z 601.252,A -85,B 0,C 180,E1 -13758.331,E2 -13758.331} C_VEL
LIN {X 0,Y 346.876,Z 608.423,A -85,B 0,C 180,E1 -13760.083,E2 -13760.083} C_VEL
LIN {X 0,Y 346.493,Z 614.136,A -85,B 0,C 180,E1 -13761.838,E2 -13761.838} C_VEL
LIN {X 0,Y 346.25,Z 619.573,A -85,B 0,C 180,E1 -13764.031,E2 -13764.031} C_VEL
LIN {X 0,Y 346.234,Z 622.023,A -85,B 0,C 180,E1 -13765.343,E2 -13765.343} C_VEL
LIN {X 0,Y 346.195,Z 623.704,A -85,B 0,C 180,E1 -13766.508,E2 -13766.508} C_VEL
LIN {X 0,Y 346.296,Z 625.854,A -85,B 0,C 180,E1 -13768.837,E2 -13768.837} C_VEL
LIN {X 0,Y 346.316,Z 626.285,A -85,B 0,C 180,E1 -13770,E2 -13770} C_VEL
LIN {X 0,Y 346.257,Z 626.313,A -85,B 0,C 180,E1 -13771.163,E2 -13771.163} C_VEL
LIN {X 0,Y 346.167,Z 625.209,A -85,B 0,C 180,E1 -13773.492,E2 -13773.492} C_VEL
LIN {X 0,Y 346.196,Z 624.033,A -85,B 0,C 180,E1 -13774.658,E2 -13774.658} C_VEL
LIN {X 0,Y 346.34,Z 620.425,A -85,B 0,C 180,E1 -13776.993,E2 -13776.993} C_VEL
LIN {X 0,Y 346.673,Z 616.546,A -85,B 0,C 180,E1 -13778.745,E2 -13778.745} C_VEL
LIN {X 0,Y 347.216,Z 611.556,A -85,B 0,C 180,E1 -13780.496,E2 -13780.496} C_VEL
LIN {X 0,Y 347.995,Z 605.309,A -85,B 0,C 180,E1 -13782.242,E2 -13782.242} C_VEL
LIN {X 0,Y 349.19,Z 597.539,A -85,B 0,C 180,E1 -13783.976,E2 -13783.976} C_VEL
LIN {X 0,Y 350.393,Z 587.991,A -85,B 0,C 180,E1 -13785.686,E2 -13785.686} C_VEL
LIN {X 0,Y 351.816,Z 577.857,A -85,B 0,C 180,E1 -13787.136,E2 -13787.136} C_VEL
LIN {X 0,Y 353.353,Z 566.582,A -85,B 0,C 180,E1 -13788.405,E2 -13788.405} C_VEL
LIN {X 0,Y 354.651,Z 555.561,A -85,B 0,C 180,E1 -13789.385,E2 -13789.385} C_VEL
LIN {X 0,Y 355.962,Z 543.349,A -85,B 0,C 180,E1 -13790.213,E2 -13790.213} C_VEL
LIN {X 0,Y 356.946,Z 530.52,A -85,B 0,C 180,E1 -13790.832,E2 -13790.832} C_VEL
LIN {X 0,Y 357.558,Z 516.974,A -85,B 0,C 180,E1 -13791.247,E2 -13791.247} C_VEL
LIN {X 0,Y 358.849,Z 451.255,A -85,B 0,C 180,E1 -13792.583,E2 -13792.583} C_VEL
LIN {X 0,Y 355.412,Z 430.264,A -85,B 0,C 180,E1 -13793.309,E2 -13793.309} C_VEL
LIN {X 0,Y 351.976,Z 412.723,A -85,B 0,C 180,E1 -13793.995,E2 -13793.995} C_VEL
LIN {X 0,Y 353.165,Z 402.473,A -85,B 0,C 180,E1 -13796.427,E2 -13796.427} C_VEL
LIN {X 0,Y 351.267,Z 392.788,A -85,B 0,C 180,E1 -13799.024,E2 -13799.024} C_VEL
LIN {X 0,Y 348.399,Z 380.686,A -85,B 0,C 180,E1 -13802.474,E2 -13802.474} C_VEL
LIN {X 0,Y 347.784,Z 378.164,A -85,B 0,C 180,E1 -13803.228,E2 -13803.228} C_VEL
LIN {X 0,Y 347.769,Z 378.168,A -85,B 0,C 180,E1 -13806.065,E2 -13806.065} C_VEL
LIN {X 0,Y 347.749,Z 378.166,A -85,B 0,C 180,E1 -13808.792,E2 -13808.792} C_VEL
LIN {X 0,Y 347.748,Z 378.166,A -85,B 0,C 180,E1 -13811.829,E2 -13811.829} C_VEL
LIN {X 0,Y 347.793,Z 378.157,A -85,B 0,C 180,E1 -13815.011,E2 -13815.011} C_VEL
LIN {X 0,Y 347.782,Z 378.158,A -85,B 0,C 180,E1 -13818.39,E2 -13818.39} C_VEL
LIN {X 0,Y 347.771,Z 378.162,A -85,B 0,C 180,E1 -13822.01,E2 -13822.01} C_VEL
LIN {X 0,Y 347.739,Z 378.169,A -85,B 0,C 180,E1 -13825.536,E2 -13825.536} C_VEL
LIN {X 0,Y 347.758,Z 378.164,A -85,B 0,C 180,E1 -13829.653,E2 -13829.653} C_VEL
LIN {X 0,Y 347.846,Z 378.153,A -85,B 0,C 180,E1 -13832.744,E2 -13832.744} C_VEL
LIN {X 0,Y 347.781,Z 378.148,A -85,B 0,C 180,E1 -13836.162,E2 -13836.162} C_VEL
LIN {X 0,Y 347.81,Z 378.155,A -85,B 0,C 180,E1 -13839.909,E2 -13839.909} C_VEL
LIN {X 0,Y 347.859,Z 378.151,A -85,B 0,C 180,E1 -13842.359,E2 -13842.359} C_VEL
LIN {X 0,Y 347.89,Z 378.147,A -85,B 0,C 180,E1 -13845.971,E2 -13845.971} C_VEL
LIN {X 0,Y 347.926,Z 378.139,A -85,B 0,C 180,E1 -13849.526,E2 -13849.526} C_VEL
LIN {X 0,Y 348.066,Z 378.127,A -85,B 0,C 180,E1 -13851.875,E2 -13851.875} C_VEL
LIN {X 0,Y 348.06,Z 378.12,A -85,B 0,C 180,E1 -13854.206,E2 -13854.206} C_VEL
LIN {X 0,Y 348.201,Z 378.107,A -85,B 0,C 180,E1 -13857.687,E2 -13857.687} C_VEL
LIN {X 0,Y 348.361,Z 378.087,A -85,B 0,C 180,E1 -13860,E2 -13860} C_VEL
LIN {X 0,Y 348.201,Z 378.111,A -85,B 0,C 180,E1 -13862.314,E2 -13862.314} C_VEL
LIN {X 0,Y 348.085,Z 378.122,A -85,B 0,C 180,E1 -13866.958,E2 -13866.958} C_VEL
LIN {X 0,Y 347.922,Z 378.148,A -85,B 0,C 180,E1 -13870.475,E2 -13870.475} C_VEL
LIN {X 0,Y 347.892,Z 378.148,A -85,B 0,C 180,E1 -13874.151,E2 -13874.151} C_VEL
LIN {X 0,Y 347.885,Z 378.149,A -85,B 0,C 180,E1 -13878.291,E2 -13878.291} C_VEL
LIN {X 0,Y 347.783,Z 378.158,A -85,B 0,C 180,E1 -13881.636,E2 -13881.636} C_VEL
LIN {X 0,Y 347.807,Z 378.148,A -85,B 0,C 180,E1 -13885.109,E2 -13885.109} C_VEL
LIN {X 0,Y 347.806,Z 378.148,A -85,B 0,C 180,E1 -13887.695,E2 -13887.695} C_VEL
LIN {X 0,Y 347.759,Z 378.166,A -85,B 0,C 180,E1 -13890.347,E2 -13890.347} C_VEL
LIN {X 0,Y 347.741,Z 378.168,A -85,B 0,C 180,E1 -13894.465,E2 -13894.465} C_VEL
LIN {X 0,Y 347.773,Z 378.168,A -85,B 0,C 180,E1 -13897.99,E2 -13897.99} C_VEL
LIN {X 0,Y 347.782,Z 378.163,A -85,B 0,C 180,E1 -13901.61,E2 -13901.61} C_VEL
LIN {X 0,Y 347.797,Z 378.167,A -85,B 0,C 180,E1 -13905.013,E2 -13905.013} C_VEL
LIN {X 0,Y 347.768,Z 378.17,A -85,B 0,C 180,E1 -13908.395,E2 -13908.395} C_VEL
LIN {X 0,Y 347.779,Z 378.166,A -85,B 0,C 180,E1 -13912.011,E2 -13912.011} C_VEL
LIN {X 0,Y 347.814,Z 378.171,A -85,B 0,C 180,E1 -13914.751,E2 -13914.751} C_VEL
LIN {X 0,Y 349.231,Z 384.495,A -85,B 0,C 180,E1 -13916.844,E2 -13916.844} C_VEL
LIN {X 0,Y 357.467,Z 403.511,A -85,B 0,C 180,E1 -13917.954,E2 -13917.954} C_VEL
LIN {X 0,Y 359.386,Z 409.067,A -85,B 0,C 180,E1 -13918.229,E2 -13918.229} C_VEL
LIN {X 0,Y 359.714,Z 410.512,A -85,B 0,C 180,E1 -13918.286,E2 -13918.286} C_VEL
LIN {X 0,Y 357.876,Z 491.281,A -85,B 0,C 180,E1 -13919.942,E2 -13919.942} C_VEL
LIN {X 0,Y 357.305,Z 503.776,A -85,B 0,C 180,E1 -13920.416,E2 -13920.416} C_VEL
LIN {X 0,Y 356.415,Z 516.324,A -85,B 0,C 180,E1 -13921.112,E2 -13921.112} C_VEL
LIN {X 0,Y 355.313,Z 527.886,A -85,B 0,C 180,E1 -13921.981,E2 -13921.981} C_VEL
LIN {X 0,Y 354.293,Z 538.543,A -85,B 0,C 180,E1 -13923.03,E2 -13923.03} C_VEL
LIN {X 0,Y 352.893,Z 549.235,A -85,B 0,C 180,E1 -13924.332,E2 -13924.332} C_VEL
LIN {X 0,Y 351.552,Z 558.921,A -85,B 0,C 180,E1 -13925.807,E2 -13925.807} C_VEL
LIN {X 0,Y 350.216,Z 568.16,A -85,B 0,C 180,E1 -13927.587,E2 -13927.587} C_VEL
LIN {X 0,Y 348.979,Z 575.549,A -85,B 0,C 180,E1 -13929.365,E2 -13929.365} C_VEL
LIN {X 0,Y 348.089,Z 581.421,A -85,B 0,C 180,E1 -13931.153,E2 -13931.153} C_VEL
LIN {X 0,Y 347.434,Z 585.996,A -85,B 0,C 180,E1 -13932.944,E2 -13932.944} C_VEL
LIN {X 0,Y 346.9,Z 589.443,A -85,B 0,C 180,E1 -13934.73,E2 -13934.73} C_VEL
LIN {X 0,Y 346.547,Z 592.105,A -85,B 0,C 180,E1 -13936.769,E2 -13936.769} C_VEL
LIN {X 0,Y 346.325,Z 593.31,A -85,B 0,C 180,E1 -13938.292,E2 -13938.292} C_VEL
LIN {X 0,Y 346.164,Z 593.768,A -85,B 0,C 180,E1 -13939.472,E2 -13939.472} C_VEL
LIN {X 0,Y 346.187,Z 593.464,A -85,B 0,C 180,E1 -13941.83,E2 -13941.83} C_VEL
LIN {X 0,Y 346.358,Z 591.921,A -85,B 0,C 180,E1 -13943.867,E2 -13943.867} C_VEL
LIN {X 0,Y 346.417,Z 590.004,A -85,B 0,C 180,E1 -13945.345,E2 -13945.345} C_VEL
LIN {X 0,Y 346.69,Z 586.847,A -85,B 0,C 180,E1 -13947.095,E2 -13947.095} C_VEL
LIN {X 0,Y 346.971,Z 582.651,A -85,B 0,C 180,E1 -13948.839,E2 -13948.839} C_VEL
LIN {X 0,Y 347.449,Z 577.282,A -85,B 0,C 180,E1 -13950.579,E2 -13950.579} C_VEL
LIN {X 0,Y 348.186,Z 570.564,A -85,B 0,C 180,E1 -13952.314,E2 -13952.314} C_VEL
LIN {X 0,Y 349.042,Z 562.23,A -85,B 0,C 180,E1 -13954.041,E2 -13954.041} C_VEL
LIN {X 0,Y 349.91,Z 553.648,A -85,B 0,C 180,E1 -13955.474,E2 -13955.474} C_VEL
LIN {X 0,Y 350.968,Z 543.083,A -85,B 0,C 180,E1 -13956.9,E2 -13956.9} C_VEL
LIN {X 0,Y 351.903,Z 532.591,A -85,B 0,C 180,E1 -13958.036,E2 -13958.036} C_VEL
LIN {X 0,Y 352.756,Z 520.939,A -85,B 0,C 180,E1 -13959.026,E2 -13959.026} C_VEL
LIN {X 0,Y 353.445,Z 508.853,A -85,B 0,C 180,E1 -13959.803,E2 -13959.803} C_VEL
LIN {X 0,Y 354,Z 495.646,A -85,B 0,C 180,E1 -13960.401,E2 -13960.401} C_VEL
LIN {X 0,Y 354.313,Z 482.581,A -85,B 0,C 180,E1 -13960.753,E2 -13960.753} C_VEL
LIN {X 0,Y 355.548,Z 407.755,A -85,B 0,C 180,E1 -13962.253,E2 -13962.253} C_VEL
LIN {X 0,Y 353.517,Z 397.647,A -85,B 0,C 180,E1 -13962.577,E2 -13962.577} C_VEL
LIN {X 0,Y 348.969,Z 383.688,A -85,B 0,C 180,E1 -13963.14,E2 -13963.14} C_VEL
LIN {X 0,Y 347.895,Z 378.151,A -85,B 0,C 180,E1 -13964.879,E2 -13964.879} C_VEL
LIN {X 0,Y 347.84,Z 378.158,A -85,B 0,C 180,E1 -13966.269,E2 -13966.269} C_VEL
LIN {X 0,Y 347.187,Z 378.243,A -85,B 0,C 180,E1 -13967.236,E2 -13967.236} C_VEL
LIN {X 0,Y 344.303,Z 378.602,A -85,B 0,C 180,E1 -13968.807,E2 -13968.807} C_VEL
LIN {X 0,Y 341.853,Z 378.902,A -85,B 0,C 180,E1 -13970.079,E2 -13970.079} C_VEL
LIN {X 0,Y 340.811,Z 379.03,A -85,B 0,C 180,E1 -13971.064,E2 -13971.064} C_VEL
LIN {X 0,Y 340.731,Z 379.039,A -85,B 0,C 180,E1 -13971.398,E2 -13971.398} C_VEL
LIN {X 0,Y 340.769,Z 379.035,A -85,B 0,C 180,E1 -13974.843,E2 -13974.843} C_VEL
LIN {X 0,Y 340.782,Z 379.032,A -85,B 0,C 180,E1 -13977.525,E2 -13977.525} C_VEL
LIN {X 0,Y 340.706,Z 379.043,A -85,B 0,C 180,E1 -13981.043,E2 -13981.043} C_VEL
LIN {X 0,Y 340.719,Z 379.04,A -85,B 0,C 180,E1 -13985.278,E2 -13985.278} C_VEL
LIN {X 0,Y 340.711,Z 379.047,A -85,B 0,C 180,E1 -13988.385,E2 -13988.385} C_VEL
LIN {X 0,Y 340.699,Z 379.045,A -85,B 0,C 180,E1 -13992.044,E2 -13992.044} C_VEL
LIN {X 0,Y 340.721,Z 379.04,A -85,B 0,C 180,E1 -13995.467,E2 -13995.467} C_VEL
LIN {X 0,Y 340.723,Z 379.042,A -85,B 0,C 180,E1 -13998.695,E2 -13998.695} C_VEL
LIN {X 0,Y 340.738,Z 379.039,A -85,B 0,C 180,E1 -14001.773,E2 -14001.773} C_VEL
LIN {X 0,Y 340.719,Z 379.039,A -85,B 0,C 180,E1 -14005.594,E2 -14005.594} C_VEL
LIN {X 0,Y 340.693,Z 379.044,A -85,B 0,C 180,E1 -14008.954,E2 -14008.954} C_VEL
LIN {X 0,Y 340.798,Z 379.03,A -85,B 0,C 180,E1 -14013.019,E2 -14013.019} C_VEL
LIN {X 0,Y 340.726,Z 379.04,A -85,B 0,C 180,E1 -14016.926,E2 -14016.926} C_VEL
LIN {X 0,Y 340.794,Z 379.032,A -85,B 0,C 180,E1 -14020.733,E2 -14020.733} C_VEL
LIN {X 0,Y 340.78,Z 379.031,A -85,B 0,C 180,E1 -14023.218,E2 -14023.218} C_VEL
LIN {X 0,Y 340.84,Z 379.025,A -85,B 0,C 180,E1 -14026.89,E2 -14026.89} C_VEL
LIN {X 0,Y 340.923,Z 379.017,A -85,B 0,C 180,E1 -14030.507,E2 -14030.507} C_VEL
LIN {X 0,Y 341.068,Z 378.996,A -85,B 0,C 180,E1 -14032.898,E2 -14032.898} C_VEL
LIN {X 0,Y 341.163,Z 378.986,A -85,B 0,C 180,E1 -14037.638,E2 -14037.638} C_VEL
LIN {X 0,Y 341.31,Z 378.971,A -85,B 0,C 180,E1 -14040,E2 -14040} C_VEL
LIN {X 0,Y 341.163,Z 378.988,A -85,B 0,C 180,E1 -14042.361,E2 -14042.361} C_VEL
LIN {X 0,Y 341.068,Z 378.997,A -85,B 0,C 180,E1 -14047.102,E2 -14047.102} C_VEL
LIN {X 0,Y 340.868,Z 379.022,A -85,B 0,C 180,E1 -14050.694,E2 -14050.694} C_VEL
LIN {X 0,Y 340.856,Z 379.026,A -85,B 0,C 180,E1 -14054.325,E2 -14054.325} C_VEL
LIN {X 0,Y 340.832,Z 379.028,A -85,B 0,C 180,E1 -14058.467,E2 -14058.467} C_VEL
LIN {X 0,Y 340.747,Z 379.041,A -85,B 0,C 180,E1 -14061.857,E2 -14061.857} C_VEL
LIN {X 0,Y 340.766,Z 379.037,A -85,B 0,C 180,E1 -14065.665,E2 -14065.665} C_VEL
LIN {X 0,Y 340.722,Z 379.042,A -85,B 0,C 180,E1 -14068.321,E2 -14068.321} C_VEL
LIN {X 0,Y 340.691,Z 379.044,A -85,B 0,C 180,E1 -14071.045,E2 -14071.045} C_VEL
LIN {X 0,Y 340.713,Z 379.042,A -85,B 0,C 180,E1 -14075.279,E2 -14075.279} C_VEL
LIN {X 0,Y 340.713,Z 379.043,A -85,B 0,C 180,E1 -14078.388,E2 -14078.388} C_VEL
LIN {X 0,Y 340.721,Z 379.041,A -85,B 0,C 180,E1 -14081.304,E2 -14081.304} C_VEL
LIN {X 0,Y 340.718,Z 379.041,A -85,B 0,C 180,E1 -14084.533,E2 -14084.533} C_VEL
LIN {X 0,Y 340.715,Z 379.046,A -85,B 0,C 180,E1 -14087.951,E2 -14087.951} C_VEL
LIN {X 0,Y 340.73,Z 379.044,A -85,B 0,C 180,E1 -14091.773,E2 -14091.773} C_VEL
LIN {X 0,Y 340.721,Z 379.044,A -85,B 0,C 180,E1 -14095.596,E2 -14095.596} C_VEL
LIN {X 0,Y 340.77,Z 379.109,A -85,B 0,C 180,E1 -14099.103,E2 -14099.103} C_VEL
LIN {X 0,Y 343.244,Z 390.988,A -85,B 0,C 180,E1 -14102.238,E2 -14102.238} C_VEL
LIN {X 0,Y 344.423,Z 397.437,A -85,B 0,C 180,E1 -14103.874,E2 -14103.874} C_VEL
LIN {X 0,Y 344.318,Z 401.905,A -85,B 0,C 180,E1 -14104.943,E2 -14104.943} C_VEL
LIN {X 0,Y 343.114,Z 412.988,A -85,B 0,C 180,E1 -14107.523,E2 -14107.523} C_VEL
LIN {X 0,Y 348.324,Z 452.336,A -85,B 0,C 180,E1 -14108.664,E2 -14108.664} C_VEL
LIN {X 0,Y 347.097,Z 521.479,A -85,B 0,C 180,E1 -14110.098,E2 -14110.098} C_VEL
LIN {X 0,Y 346.478,Z 534.853,A -85,B 0,C 180,E1 -14110.601,E2 -14110.601} C_VEL
LIN {X 0,Y 345.576,Z 547.651,A -85,B 0,C 180,E1 -14111.319,E2 -14111.319} C_VEL
LIN {X 0,Y 344.647,Z 559.017,A -85,B 0,C 180,E1 -14112.189,E2 -14112.189} C_VEL
LIN {X 0,Y 343.386,Z 570.733,A -85,B 0,C 180,E1 -14113.35,E2 -14113.35} C_VEL
LIN {X 0,Y 342.482,Z 580.213,A -85,B 0,C 180,E1 -14114.528,E2 -14114.528} C_VEL
LIN {X 0,Y 341.609,Z 589.93,A -85,B 0,C 180,E1 -14116.011,E2 -14116.011} C_VEL
LIN {X 0,Y 340.781,Z 597.872,A -85,B 0,C 180,E1 -14117.494,E2 -14117.494} C_VEL
LIN {X 0,Y 339.986,Z 605.611,A -85,B 0,C 180,E1 -14119.278,E2 -14119.278} C_VEL
LIN {X 0,Y 339.54,Z 611.834,A -85,B 0,C 180,E1 -14121.07,E2 -14121.07} C_VEL
LIN {X 0,Y 339.249,Z 616.763,A -85,B 0,C 180,E1 -14122.86,E2 -14122.86} C_VEL
LIN {X 0,Y 339.13,Z 620.298,A -85,B 0,C 180,E1 -14124.511,E2 -14124.511} C_VEL
LIN {X 0,Y 339.118,Z 623.296,A -85,B 0,C 180,E1 -14126.436,E2 -14126.436} C_VEL
LIN {X 0,Y 339.2,Z 625.482,A -85,B 0,C 180,E1 -14128.813,E2 -14128.813} C_VEL
LIN {X 0,Y 339.224,Z 625.943,A -85,B 0,C 180,E1 -14130,E2 -14130} C_VEL
LIN {X 0,Y 339.159,Z 625.986,A -85,B 0,C 180,E1 -14131.187,E2 -14131.187} C_VEL
LIN {X 0,Y 339.091,Z 624.916,A -85,B 0,C 180,E1 -14133.565,E2 -14133.565} C_VEL
LIN {X 0,Y 339.094,Z 623.773,A -85,B 0,C 180,E1 -14134.755,E2 -14134.755} C_VEL
LIN {X 0,Y 339.129,Z 622.192,A -85,B 0,C 180,E1 -14135.947,E2 -14135.947} C_VEL
LIN {X 0,Y 339.38,Z 619.042,A -85,B 0,C 180,E1 -14137.736,E2 -14137.736} C_VEL
LIN {X 0,Y 339.771,Z 614.845,A -85,B 0,C 180,E1 -14139.525,E2 -14139.525} C_VEL
LIN {X 0,Y 340.534,Z 608.478,A -85,B 0,C 180,E1 -14141.608,E2 -14141.608} C_VEL
LIN {X 0,Y 341.654,Z 601.573,A -85,B 0,C 180,E1 -14143.38,E2 -14143.38} C_VEL
LIN {X 0,Y 342.864,Z 592.963,A -85,B 0,C 180,E1 -14145.15,E2 -14145.15} C_VEL
LIN {X 0,Y 344.144,Z 584.16,A -85,B 0,C 180,E1 -14146.612,E2 -14146.612} C_VEL
LIN {X 0,Y 345.575,Z 574.522,A -85,B 0,C 180,E1 -14147.914,E2 -14147.914} C_VEL
LIN {X 0,Y 347.005,Z 564.006,A -85,B 0,C 180,E1 -14149.061,E2 -14149.061} C_VEL
LIN {X 0,Y 348.463,Z 552.363,A -85,B 0,C 180,E1 -14150.051,E2 -14150.051} C_VEL
LIN {X 0,Y 349.664,Z 540.299,A -85,B 0,C 180,E1 -14150.824,E2 -14150.824} C_VEL
LIN {X 0,Y 350.634,Z 527.202,A -85,B 0,C 180,E1 -14151.418,E2 -14151.418} C_VEL
LIN {X 0,Y 351.155,Z 514.639,A -85,B 0,C 180,E1 -14151.77,E2 -14151.77} C_VEL
LIN {X 0,Y 352.441,Z 452.303,A -85,B 0,C 180,E1 -14153.055,E2 -14153.055} C_VEL
LIN {X 0,Y 349.129,Z 431.947,A -85,B 0,C 180,E1 -14153.778,E2 -14153.778} C_VEL
LIN {X 0,Y 345.274,Z 412.38,A -85,B 0,C 180,E1 -14154.568,E2 -14154.568} C_VEL
LIN {X 0,Y 346.275,Z 404.315,A -85,B 0,C 180,E1 -14156.519,E2 -14156.519} C_VEL
LIN {X 0,Y 344.764,Z 396.048,A -85,B 0,C 180,E1 -14158.771,E2 -14158.771} C_VEL
LIN {X 0,Y 341.898,Z 383.84,A -85,B 0,C 180,E1 -14162.306,E2 -14162.306} C_VEL
LIN {X 0,Y 340.73,Z 379.043,A -85,B 0,C 180,E1 -14163.797,E2 -14163.797} C_VEL
LIN {X 0,Y 340.703,Z 379.046,A -85,B 0,C 180,E1 -14166.741,E2 -14166.741} C_VEL
LIN {X 0,Y 340.685,Z 379.046,A -85,B 0,C 180,E1 -14170.246,E2 -14170.246} C_VEL
LIN {X 0,Y 340.673,Z 379.047,A -85,B 0,C 180,E1 -14173.777,E2 -14173.777} C_VEL
LIN {X 0,Y 340.737,Z 379.036,A -85,B 0,C 180,E1 -14177.105,E2 -14177.105} C_VEL
LIN {X 0,Y 340.73,Z 379.038,A -85,B 0,C 180,E1 -14180.252,E2 -14180.252} C_VEL
LIN {X 0,Y 340.706,Z 379.045,A -85,B 0,C 180,E1 -14183.559,E2 -14183.559} C_VEL
LIN {X 0,Y 340.686,Z 379.046,A -85,B 0,C 180,E1 -14186.153,E2 -14186.153} C_VEL
LIN {X 0,Y 340.769,Z 379.034,A -85,B 0,C 180,E1 -14190.332,E2 -14190.332} C_VEL
LIN {X 0,Y 340.799,Z 379.027,A -85,B 0,C 180,E1 -14193.02,E2 -14193.02} C_VEL
LIN {X 0,Y 340.722,Z 379.032,A -85,B 0,C 180,E1 -14196.927,E2 -14196.927} C_VEL
LIN {X 0,Y 340.787,Z 379.029,A -85,B 0,C 180,E1 -14200.734,E2 -14200.734} C_VEL
LIN {X 0,Y 340.78,Z 379.037,A -85,B 0,C 180,E1 -14203.218,E2 -14203.218} C_VEL
LIN {X 0,Y 340.839,Z 379.028,A -85,B 0,C 180,E1 -14206.891,E2 -14206.891} C_VEL
LIN {X 0,Y 340.923,Z 379.013,A -85,B 0,C 180,E1 -14210.508,E2 -14210.508} C_VEL
LIN {X 0,Y 341.068,Z 378.998,A -85,B 0,C 180,E1 -14212.898,E2 -14212.898} C_VEL
LIN {X 0,Y 341.163,Z 378.983,A -85,B 0,C 180,E1 -14217.639,E2 -14217.639} C_VEL
LIN {X 0,Y 341.31,Z 378.966,A -85,B 0,C 180,E1 -14220,E2 -14220} C_VEL
LIN {X 0,Y 341.163,Z 378.988,A -85,B 0,C 180,E1 -14222.362,E2 -14222.362} C_VEL
LIN {X 0,Y 341.053,Z 378.997,A -85,B 0,C 180,E1 -14227.103,E2 -14227.103} C_VEL
LIN {X 0,Y 340.864,Z 379.027,A -85,B 0,C 180,E1 -14230.694,E2 -14230.694} C_VEL
LIN {X 0,Y 340.857,Z 379.025,A -85,B 0,C 180,E1 -14234.326,E2 -14234.326} C_VEL
LIN {X 0,Y 340.832,Z 379.03,A -85,B 0,C 180,E1 -14238.468,E2 -14238.468} C_VEL
LIN {X 0,Y 340.748,Z 379.035,A -85,B 0,C 180,E1 -14241.858,E2 -14241.858} C_VEL
LIN {X 0,Y 340.767,Z 379.02,A -85,B 0,C 180,E1 -14245.665,E2 -14245.665} C_VEL
LIN {X 0,Y 340.736,Z 379.034,A -85,B 0,C 180,E1 -14248.321,E2 -14248.321} C_VEL
LIN {X 0,Y 340.699,Z 379.04,A -85,B 0,C 180,E1 -14251.045,E2 -14251.045} C_VEL
LIN {X 0,Y 340.715,Z 379.043,A -85,B 0,C 180,E1 -14255.28,E2 -14255.28} C_VEL
LIN {X 0,Y 340.715,Z 379.046,A -85,B 0,C 180,E1 -14258.389,E2 -14258.389} C_VEL
LIN {X 0,Y 340.723,Z 379.045,A -85,B 0,C 180,E1 -14261.305,E2 -14261.305} C_VEL
LIN {X 0,Y 340.737,Z 379.048,A -85,B 0,C 180,E1 -14264.531,E2 -14264.531} C_VEL
LIN {X 0,Y 340.733,Z 379.049,A -85,B 0,C 180,E1 -14267.949,E2 -14267.949} C_VEL
LIN {X 0,Y 340.741,Z 379.044,A -85,B 0,C 180,E1 -14271.775,E2 -14271.775} C_VEL
LIN {X 0,Y 340.769,Z 379.127,A -85,B 0,C 180,E1 -14274.275,E2 -14274.275} C_VEL
LIN {X 0,Y 342.125,Z 384.909,A -85,B 0,C 180,E1 -14276.227,E2 -14276.227} C_VEL
LIN {X 0,Y 351.501,Z 406.282,A -85,B 0,C 180,E1 -14277.53,E2 -14277.53} C_VEL
LIN {X 0,Y 353.278,Z 411.479,A -85,B 0,C 180,E1 -14277.792,E2 -14277.792} C_VEL
LIN {X 0,Y 351.442,Z 491.574,A -85,B 0,C 180,E1 -14279.469,E2 -14279.469} C_VEL
LIN {X 0,Y 350.825,Z 504.048,A -85,B 0,C 180,E1 -14279.947,E2 -14279.947} C_VEL
LIN {X 0,Y 349.869,Z 517.06,A -85,B 0,C 180,E1 -14280.684,E2 -14280.684} C_VEL
LIN {X 0,Y 348.719,Z 528.497,A -85,B 0,C 180,E1 -14281.568,E2 -14281.568} C_VEL
LIN {X 0,Y 347.559,Z 539.841,A -85,B 0,C 180,E1 -14282.718,E2 -14282.718} C_VEL
LIN {X 0,Y 346.038,Z 550.836,A -85,B 0,C 180,E1 -14284.11,E2 -14284.11} C_VEL
LIN {X 0,Y 344.645,Z 560.228,A -85,B 0,C 180,E1 -14285.611,E2 -14285.611} C_VEL
LIN {X 0,Y 343.259,Z 569.294,A -85,B 0,C 180,E1 -14287.425,E2 -14287.425} C_VEL
LIN {X 0,Y 342,Z 576.528,A -85,B 0,C 180,E1 -14289.239,E2 -14289.239} C_VEL
LIN {X 0,Y 340.979,Z 582.798,A -85,B 0,C 180,E1 -14291.272,E2 -14291.272} C_VEL
LIN {X 0,Y 340.262,Z 587.321,A -85,B 0,C 180,E1 -14293.192,E2 -14293.192} C_VEL
LIN {X 0,Y 339.89,Z 589.57,A -85,B 0,C 180,E1 -14294.407,E2 -14294.407} C_VEL
LIN {X 0,Y 339.486,Z 592.477,A -85,B 0,C 180,E1 -14296.656,E2 -14296.656} C_VEL
LIN {X 0,Y 339.262,Z 593.563,A -85,B 0,C 180,E1 -14298.045,E2 -14298.045} C_VEL
LIN {X 0,Y 339.103,Z 594.083,A -85,B 0,C 180,E1 -14299.25,E2 -14299.25} C_VEL
LIN {X 0,Y 339.103,Z 593.85,A -85,B 0,C 180,E1 -14301.658,E2 -14301.658} C_VEL
LIN {X 0,Y 339.275,Z 592.229,A -85,B 0,C 180,E1 -14303.891,E2 -14303.891} C_VEL
LIN {X 0,Y 339.34,Z 590.522,A -85,B 0,C 180,E1 -14305.248,E2 -14305.248} C_VEL
LIN {X 0,Y 339.582,Z 587.44,A -85,B 0,C 180,E1 -14307.034,E2 -14307.034} C_VEL
LIN {X 0,Y 339.889,Z 583.318,A -85,B 0,C 180,E1 -14308.815,E2 -14308.815} C_VEL
LIN {X 0,Y 340.374,Z 578.032,A -85,B 0,C 180,E1 -14310.592,E2 -14310.592} C_VEL
LIN {X 0,Y 341.114,Z 571.407,A -85,B 0,C 180,E1 -14312.362,E2 -14312.362} C_VEL
LIN {X 0,Y 342.004,Z 563.2,A -85,B 0,C 180,E1 -14314.124,E2 -14314.124} C_VEL
LIN {X 0,Y 342.874,Z 554.787,A -85,B 0,C 180,E1 -14315.587,E2 -14315.587} C_VEL
LIN {X 0,Y 343.99,Z 544.383,A -85,B 0,C 180,E1 -14317.041,E2 -14317.041} C_VEL
LIN {X 0,Y 344.942,Z 534.1,A -85,B 0,C 180,E1 -14318.199,E2 -14318.199} C_VEL
LIN {X 0,Y 345.799,Z 522.853,A -85,B 0,C 180,E1 -14319.21,E2 -14319.21} C_VEL
LIN {X 0,Y 346.533,Z 511.331,A -85,B 0,C 180,E1 -14320,E2 -14320} C_VEL
LIN {X 0,Y 347.136,Z 498.095,A -85,B 0,C 180,E1 -14320.646,E2 -14320.646} C_VEL
LIN {X 0,Y 347.488,Z 485.181,A -85,B 0,C 180,E1 -14321.04,E2 -14321.04} C_VEL
LIN {X 0,Y 348.845,Z 408.679,A -85,B 0,C 180,E1 -14322.603,E2 -14322.603} C_VEL
LIN {X 0,Y 346.803,Z 399.063,A -85,B 0,C 180,E1 -14322.925,E2 -14322.925} C_VEL
LIN {X 0,Y 341.833,Z 384.019,A -85,B 0,C 180,E1 -14323.553,E2 -14323.553} C_VEL
LIN {X 0,Y 340.839,Z 379.031,A -85,B 0,C 180,E1 -14325.127,E2 -14325.127} C_VEL
LIN {X 0,Y 340.842,Z 379.031,A -85,B 0,C 180,E1 -14328.466,E2 -14328.466} C_VEL
LIN {X 0,Y 340.731,Z 379.039,A -85,B 0,C 180,E1 -14331.398,E2 -14331.398} C_VEL
LIN {X 0,Y 340.085,Z 379.125,A -85,B 0,C 180,E1 -14332.385,E2 -14332.385} C_VEL
LIN {X 0,Y 337.259,Z 379.475,A -85,B 0,C 180,E1 -14333.991,E2 -14333.991} C_VEL
LIN {X 0,Y 334.851,Z 379.775,A -85,B 0,C 180,E1 -14335.291,E2 -14335.291} C_VEL
LIN {X 0,Y 333.81,Z 379.904,A -85,B 0,C 180,E1 -14336.297,E2 -14336.297} C_VEL
LIN {X 0,Y 333.722,Z 379.911,A -85,B 0,C 180,E1 -14336.638,E2 -14336.638} C_VEL
LIN {X 0,Y 333.699,Z 379.92,A -85,B 0,C 180,E1 -14340.361,E2 -14340.361} C_VEL
LIN {X 0,Y 333.675,Z 379.921,A -85,B 0,C 180,E1 -14344.658,E2 -14344.658} C_VEL
LIN {X 0,Y 333.653,Z 379.921,A -85,B 0,C 180,E1 -14347.65,E2 -14347.65} C_VEL
LIN {X 0,Y 333.646,Z 379.922,A -85,B 0,C 180,E1 -14350.766,E2 -14350.766} C_VEL
LIN {X 0,Y 333.643,Z 379.927,A -85,B 0,C 180,E1 -14354.258,E2 -14354.258} C_VEL
LIN {X 0,Y 333.693,Z 379.914,A -85,B 0,C 180,E1 -14357.626,E2 -14357.626} C_VEL
LIN {X 0,Y 333.681,Z 379.917,A -85,B 0,C 180,E1 -14361.194,E2 -14361.194} C_VEL
LIN {X 0,Y 333.682,Z 379.914,A -85,B 0,C 180,E1 -14365.225,E2 -14365.225} C_VEL
LIN {X 0,Y 333.627,Z 379.929,A -85,B 0,C 180,E1 -14368.221,E2 -14368.221} C_VEL
LIN {X 0,Y 333.685,Z 379.916,A -85,B 0,C 180,E1 -14371.025,E2 -14371.025} C_VEL
LIN {X 0,Y 333.73,Z 379.911,A -85,B 0,C 180,E1 -14373.753,E2 -14373.753} C_VEL
LIN {X 0,Y 333.714,Z 379.915,A -85,B 0,C 180,E1 -14377.913,E2 -14377.913} C_VEL
LIN {X 0,Y 333.789,Z 379.904,A -85,B 0,C 180,E1 -14381.589,E2 -14381.589} C_VEL
LIN {X 0,Y 333.802,Z 379.901,A -85,B 0,C 180,E1 -14385.576,E2 -14385.576} C_VEL
LIN {X 0,Y 333.831,Z 379.898,A -85,B 0,C 180,E1 -14389.078,E2 -14389.078} C_VEL
LIN {X 0,Y 334.018,Z 379.875,A -85,B 0,C 180,E1 -14392.747,E2 -14392.747} C_VEL
LIN {X 0,Y 333.805,Z 379.898,A -85,B 0,C 180,E1 -14395.169,E2 -14395.169} C_VEL
LIN {X 0,Y 334.1,Z 379.865,A -85,B 0,C 180,E1 -14397.588,E2 -14397.588} C_VEL
LIN {X 0,Y 334.26,Z 379.85,A -85,B 0,C 180,E1 -14400,E2 -14400} C_VEL
LIN {X 0,Y 334.101,Z 379.867,A -85,B 0,C 180,E1 -14402.411,E2 -14402.411} C_VEL
LIN {X 0,Y 334.018,Z 379.875,A -85,B 0,C 180,E1 -14407.252,E2 -14407.252} C_VEL
LIN {X 0,Y 333.831,Z 379.898,A -85,B 0,C 180,E1 -14410.922,E2 -14410.922} C_VEL
LIN {X 0,Y 333.801,Z 379.903,A -85,B 0,C 180,E1 -14414.634,E2 -14414.634} C_VEL
LIN {X 0,Y 333.791,Z 379.903,A -85,B 0,C 180,E1 -14418.656,E2 -14418.656} C_VEL
LIN {X 0,Y 333.686,Z 379.919,A -85,B 0,C 180,E1 -14422.278,E2 -14422.278} C_VEL
LIN {X 0,Y 333.728,Z 379.915,A -85,B 0,C 180,E1 -14426.247,E2 -14426.247} C_VEL
LIN {X 0,Y 333.684,Z 379.917,A -85,B 0,C 180,E1 -14428.975,E2 -14428.975} C_VEL
LIN {X 0,Y 333.638,Z 379.923,A -85,B 0,C 180,E1 -14432.587,E2 -14432.587} C_VEL
LIN {X 0,Y 333.671,Z 379.922,A -85,B 0,C 180,E1 -14436.139,E2 -14436.139} C_VEL
LIN {X 0,Y 333.679,Z 379.918,A -85,B 0,C 180,E1 -14439.188,E2 -14439.188} C_VEL
LIN {X 0,Y 333.686,Z 379.917,A -85,B 0,C 180,E1 -14442.511,E2 -14442.511} C_VEL
LIN {X 0,Y 333.643,Z 379.927,A -85,B 0,C 180,E1 -14445.964,E2 -14445.964} C_VEL
LIN {X 0,Y 333.644,Z 379.923,A -85,B 0,C 180,E1 -14449.316,E2 -14449.316} C_VEL
LIN {X 0,Y 333.663,Z 379.92,A -85,B 0,C 180,E1 -14453.168,E2 -14453.168} C_VEL
LIN {X 0,Y 333.64,Z 379.925,A -85,B 0,C 180,E1 -14456.793,E2 -14456.793} C_VEL
LIN {X 0,Y 333.708,Z 379.921,A -85,B 0,C 180,E1 -14458.762,E2 -14458.762} C_VEL
LIN {X 0,Y 336.457,Z 393.17,A -85,B 0,C 180,E1 -14462.328,E2 -14462.328} C_VEL
LIN {X 0,Y 337.586,Z 399.944,A -85,B 0,C 180,E1 -14464.076,E2 -14464.076} C_VEL
LIN {X 0,Y 336.248,Z 412.691,A -85,B 0,C 180,E1 -14467.117,E2 -14467.117} C_VEL
LIN {X 0,Y 341.595,Z 452.484,A -85,B 0,C 180,E1 -14468.301,E2 -14468.301} C_VEL
LIN {X 0,Y 340.298,Z 521.483,A -85,B 0,C 180,E1 -14469.762,E2 -14469.762} C_VEL
LIN {X 0,Y 339.67,Z 534.747,A -85,B 0,C 180,E1 -14470.275,E2 -14470.275} C_VEL
LIN {X 0,Y 338.745,Z 547.487,A -85,B 0,C 180,E1 -14471.006,E2 -14471.006} C_VEL
LIN {X 0,Y 337.698,Z 559.601,A -85,B 0,C 180,E1 -14471.967,E2 -14471.967} C_VEL
LIN {X 0,Y 336.399,Z 571.147,A -85,B 0,C 180,E1 -14473.15,E2 -14473.15} C_VEL
LIN {X 0,Y 335.364,Z 581.716,A -85,B 0,C 180,E1 -14474.523,E2 -14474.523} C_VEL
LIN {X 0,Y 334.463,Z 590.935,A -85,B 0,C 180,E1 -14476.017,E2 -14476.017} C_VEL
LIN {X 0,Y 333.525,Z 600.006,A -85,B 0,C 180,E1 -14477.836,E2 -14477.836} C_VEL
LIN {X 0,Y 332.8,Z 607.301,A -85,B 0,C 180,E1 -14479.66,E2 -14479.66} C_VEL
LIN {X 0,Y 332.36,Z 613.122,A -85,B 0,C 180,E1 -14481.488,E2 -14481.488} C_VEL
LIN {X 0,Y 332.114,Z 617.695,A -85,B 0,C 180,E1 -14483.316,E2 -14483.316} C_VEL
LIN {X 0,Y 332.048,Z 621.164,A -85,B 0,C 180,E1 -14485.144,E2 -14485.144} C_VEL
LIN {X 0,Y 332.043,Z 622.885,A -85,B 0,C 180,E1 -14486.359,E2 -14486.359} C_VEL
LIN {X 0,Y 332.103,Z 625.105,A -85,B 0,C 180,E1 -14488.787,E2 -14488.787} C_VEL
LIN {X 0,Y 332.132,Z 625.6,A -85,B 0,C 180,E1 -14490,E2 -14490} C_VEL
LIN {X 0,Y 332.062,Z 625.661,A -85,B 0,C 180,E1 -14491.213,E2 -14491.213} C_VEL
LIN {X 0,Y 332.015,Z 624.624,A -85,B 0,C 180,E1 -14493.641,E2 -14493.641} C_VEL
LIN {X 0,Y 332.013,Z 622.364,A -85,B 0,C 180,E1 -14495.794,E2 -14495.794} C_VEL
LIN {X 0,Y 332.317,Z 618.838,A -85,B 0,C 180,E1 -14497.901,E2 -14497.901} C_VEL
LIN {X 0,Y 332.749,Z 614.68,A -85,B 0,C 180,E1 -14499.728,E2 -14499.728} C_VEL
LIN {X 0,Y 333.564,Z 608.355,A -85,B 0,C 180,E1 -14501.854,E2 -14501.854} C_VEL
LIN {X 0,Y 334.734,Z 601.498,A -85,B 0,C 180,E1 -14503.662,E2 -14503.662} C_VEL
LIN {X 0,Y 336.004,Z 592.977,A -85,B 0,C 180,E1 -14505.467,E2 -14505.467} C_VEL
LIN {X 0,Y 337.326,Z 584.248,A -85,B 0,C 180,E1 -14506.958,E2 -14506.958} C_VEL
LIN {X 0,Y 339.023,Z 573.528,A -85,B 0,C 180,E1 -14508.429,E2 -14508.429} C_VEL
LIN {X 0,Y 340.534,Z 562.864,A -85,B 0,C 180,E1 -14509.595,E2 -14509.595} C_VEL
LIN {X 0,Y 341.998,Z 550.933,A -85,B 0,C 180,E1 -14510.604,E2 -14510.604} C_VEL
LIN {X 0,Y 343.291,Z 538.532,A -85,B 0,C 180,E1 -14511.386,E2 -14511.386} C_VEL
LIN {X 0,Y 344.24,Z 525.72,A -85,B 0,C 180,E1 -14511.954,E2 -14511.954} C_VEL
LIN {X 0,Y 344.821,Z 512.145,A -85,B 0,C 180,E1 -14512.309,E2 -14512.309} C_VEL
LIN {X 0,Y 346.118,Z 453.7,A -85,B 0,C 180,E1 -14513.532,E2 -14513.532} C_VEL
LIN {X 0,Y 342.851,Z 433.337,A -85,B 0,C 180,E1 -14514.273,E2 -14514.273} C_VEL
LIN {X 0,Y 338.586,Z 412.067,A -85,B 0,C 180,E1 -14515.153,E2 -14515.153} C_VEL
LIN {X 0,Y 339.408,Z 405.395,A -85,B 0,C 180,E1 -14516.809,E2 -14516.809} C_VEL
LIN {X 0,Y 337.541,Z 396.063,A -85,B 0,C 180,E1 -14519.437,E2 -14519.437} C_VEL
LIN {X 0,Y 334.81,Z 384.476,A -85,B 0,C 180,E1 -14522.898,E2 -14522.898} C_VEL
LIN {X 0,Y 333.675,Z 379.923,A -85,B 0,C 180,E1 -14524.383,E2 -14524.383} C_VEL
LIN {X 0,Y 333.65,Z 379.924,A -85,B 0,C 180,E1 -14527.65,E2 -14527.65} C_VEL
LIN {X 0,Y 333.643,Z 379.921,A -85,B 0,C 180,E1 -14530.767,E2 -14530.767} C_VEL
LIN {X 0,Y 333.639,Z 379.921,A -85,B 0,C 180,E1 -14534.258,E2 -14534.258} C_VEL
LIN {X 0,Y 333.692,Z 379.915,A -85,B 0,C 180,E1 -14537.626,E2 -14537.626} C_VEL
LIN {X 0,Y 333.678,Z 379.917,A -85,B 0,C 180,E1 -14541.195,E2 -14541.195} C_VEL
LIN {X 0,Y 333.68,Z 379.919,A -85,B 0,C 180,E1 -14545.225,E2 -14545.225} C_VEL
LIN {X 0,Y 333.692,Z 379.915,A -85,B 0,C 180,E1 -14549.637,E2 -14549.637} C_VEL
LIN {X 0,Y 333.738,Z 379.91,A -85,B 0,C 180,E1 -14552.401,E2 -14552.401} C_VEL
LIN {X 0,Y 333.72,Z 379.891,A -85,B 0,C 180,E1 -14555.09,E2 -14555.09} C_VEL
LIN {X 0,Y 333.675,Z 379.922,A -85,B 0,C 180,E1 -14559.019,E2 -14559.019} C_VEL
LIN {X 0,Y 333.787,Z 379.904,A -85,B 0,C 180,E1 -14561.589,E2 -14561.589} C_VEL
LIN {X 0,Y 333.801,Z 379.901,A -85,B 0,C 180,E1 -14565.577,E2 -14565.577} C_VEL
LIN {X 0,Y 333.83,Z 379.896,A -85,B 0,C 180,E1 -14569.078,E2 -14569.078} C_VEL
LIN {X 0,Y 334.018,Z 379.878,A -85,B 0,C 180,E1 -14572.748,E2 -14572.748} C_VEL
LIN {X 0,Y 333.806,Z 379.902,A -85,B 0,C 180,E1 -14575.169,E2 -14575.169} C_VEL
LIN {X 0,Y 334.101,Z 379.863,A -85,B 0,C 180,E1 -14577.589,E2 -14577.589} C_VEL
LIN {X 0,Y 334.26,Z 379.844,A -85,B 0,C 180,E1 -14580,E2 -14580} C_VEL
LIN {X 0,Y 334.1,Z 379.867,A -85,B 0,C 180,E1 -14582.412,E2 -14582.412} C_VEL
LIN {X 0,Y 333.986,Z 379.876,A -85,B 0,C 180,E1 -14586.673,E2 -14586.673} C_VEL
LIN {X 0,Y 333.844,Z 379.897,A -85,B 0,C 180,E1 -14589.696,E2 -14589.696} C_VEL
LIN {X 0,Y 333.79,Z 379.902,A -85,B 0,C 180,E1 -14593.392,E2 -14593.392} C_VEL
LIN {X 0,Y 333.74,Z 379.907,A -85,B 0,C 180,E1 -14597.147,E2 -14597.147} C_VEL
LIN {X 0,Y 333.733,Z 379.912,A -85,B 0,C 180,E1 -14599.691,E2 -14599.691} C_VEL
LIN {X 0,Y 333.687,Z 379.918,A -85,B 0,C 180,E1 -14602.279,E2 -14602.279} C_VEL
LIN {X 0,Y 333.731,Z 379.892,A -85,B 0,C 180,E1 -14606.247,E2 -14606.247} C_VEL
LIN {X 0,Y 333.706,Z 379.916,A -85,B 0,C 180,E1 -14608.973,E2 -14608.973} C_VEL
LIN {X 0,Y 333.639,Z 379.926,A -85,B 0,C 180,E1 -14612.588,E2 -14612.588} C_VEL
LIN {X 0,Y 333.673,Z 379.922,A -85,B 0,C 180,E1 -14616.14,E2 -14616.14} C_VEL
LIN {X 0,Y 333.682,Z 379.919,A -85,B 0,C 180,E1 -14619.188,E2 -14619.188} C_VEL
LIN {X 0,Y 333.688,Z 379.913,A -85,B 0,C 180,E1 -14622.512,E2 -14622.512} C_VEL
LIN {X 0,Y 333.658,Z 379.922,A -85,B 0,C 180,E1 -14625.967,E2 -14625.967} C_VEL
LIN {X 0,Y 333.656,Z 379.929,A -85,B 0,C 180,E1 -14629.315,E2 -14629.315} C_VEL
LIN {X 0,Y 333.658,Z 379.925,A -85,B 0,C 180,E1 -14632.351,E2 -14632.351} C_VEL
LIN {X 0,Y 333.721,Z 380.106,A -85,B 0,C 180,E1 -14633.781,E2 -14633.781} C_VEL
LIN {X 0,Y 334.919,Z 385.137,A -85,B 0,C 180,E1 -14635.563,E2 -14635.563} C_VEL
LIN {X 0,Y 344.564,Z 406.686,A -85,B 0,C 180,E1 -14636.95,E2 -14636.95} C_VEL
LIN {X 0,Y 346.907,Z 412.658,A -85,B 0,C 180,E1 -14637.288,E2 -14637.288} C_VEL
LIN {X 0,Y 345.051,Z 491.55,A -85,B 0,C 180,E1 -14638.967,E2 -14638.967} C_VEL
LIN {X 0,Y 344.452,Z 503.398,A -85,B 0,C 180,E1 -14639.416,E2 -14639.416} C_VEL
LIN {X 0,Y 343.457,Z 516.666,A -85,B 0,C 180,E1 -14640.166,E2 -14640.166} C_VEL
LIN {X 0,Y 342.315,Z 527.435,A -85,B 0,C 180,E1 -14640.986,E2 -14640.986} C_VEL
LIN {X 0,Y 341.142,Z 538.694,A -85,B 0,C 180,E1 -14642.11,E2 -14642.11} C_VEL
LIN {X 0,Y 339.638,Z 549.191,A -85,B 0,C 180,E1 -14643.419,E2 -14643.419} C_VEL
LIN {X 0,Y 338.307,Z 558.096,A -85,B 0,C 180,E1 -14644.795,E2 -14644.795} C_VEL
LIN {X 0,Y 337.017,Z 566.237,A -85,B 0,C 180,E1 -14646.333,E2 -14646.333} C_VEL
LIN {X 0,Y 335.606,Z 574.148,A -85,B 0,C 180,E1 -14648.18,E2 -14648.18} C_VEL
LIN {X 0,Y 334.641,Z 579.496,A -85,B 0,C 180,E1 -14649.725,E2 -14649.725} C_VEL
LIN {X 0,Y 333.78,Z 584.65,A -85,B 0,C 180,E1 -14651.589,E2 -14651.589} C_VEL
LIN {X 0,Y 333.095,Z 588.613,A -85,B 0,C 180,E1 -14653.451,E2 -14653.451} C_VEL
LIN {X 0,Y 332.616,Z 591.509,A -85,B 0,C 180,E1 -14655.312,E2 -14655.312} C_VEL
LIN {X 0,Y 332.425,Z 592.862,A -85,B 0,C 180,E1 -14656.553,E2 -14656.553} C_VEL
LIN {X 0,Y 332.05,Z 594.378,A -85,B 0,C 180,E1 -14659.019,E2 -14659.019} C_VEL
LIN {X 0,Y 331.986,Z 594.515,A -85,B 0,C 180,E1 -14660.25,E2 -14660.25} C_VEL
LIN {X 0,Y 332.102,Z 593.572,A -85,B 0,C 180,E1 -14662.705,E2 -14662.705} C_VEL
LIN {X 0,Y 332.184,Z 592.525,A -85,B 0,C 180,E1 -14663.928,E2 -14663.928} C_VEL
LIN {X 0,Y 332.243,Z 591.042,A -85,B 0,C 180,E1 -14665.146,E2 -14665.146} C_VEL
LIN {X 0,Y 332.479,Z 588.032,A -85,B 0,C 180,E1 -14666.971,E2 -14666.971} C_VEL
LIN {X 0,Y 332.795,Z 583.986,A -85,B 0,C 180,E1 -14668.79,E2 -14668.79} C_VEL
LIN {X 0,Y 333.417,Z 577.779,A -85,B 0,C 180,E1 -14670.906,E2 -14670.906} C_VEL
LIN {X 0,Y 334.209,Z 571.024,A -85,B 0,C 180,E1 -14672.712,E2 -14672.712} C_VEL
LIN {X 0,Y 335.123,Z 562.628,A -85,B 0,C 180,E1 -14674.51,E2 -14674.51} C_VEL
LIN {X 0,Y 336.073,Z 553.991,A -85,B 0,C 180,E1 -14676.002,E2 -14676.002} C_VEL
LIN {X 0,Y 337.224,Z 543.357,A -85,B 0,C 180,E1 -14677.484,E2 -14677.484} C_VEL
LIN {X 0,Y 338.237,Z 532.769,A -85,B 0,C 180,E1 -14678.664,E2 -14678.664} C_VEL
LIN {X 0,Y 339.113,Z 520.948,A -85,B 0,C 180,E1 -14679.694,E2 -14679.694} C_VEL
LIN {X 0,Y 339.905,Z 508.64,A -85,B 0,C 180,E1 -14680.498,E2 -14680.498} C_VEL
LIN {X 0,Y 340.449,Z 495.971,A -85,B 0,C 180,E1 -14681.083,E2 -14681.083} C_VEL
LIN {X 0,Y 340.781,Z 482.627,A -85,B 0,C 180,E1 -14681.449,E2 -14681.449} C_VEL
LIN {X 0,Y 342.114,Z 409.469,A -85,B 0,C 180,E1 -14682.969,E2 -14682.969} C_VEL
LIN {X 0,Y 340.237,Z 400.819,A -85,B 0,C 180,E1 -14683.27,E2 -14683.27} C_VEL
LIN {X 0,Y 334.659,Z 384.302,A -85,B 0,C 180,E1 -14683.997,E2 -14683.997} C_VEL
LIN {X 0,Y 333.782,Z 379.912,A -85,B 0,C 180,E1 -14685.455,E2 -14685.455} C_VEL
LIN {X 0,Y 333.801,Z 379.907,A -85,B 0,C 180,E1 -14688.655,E2 -14688.655} C_VEL
LIN {X 0,Y 333.696,Z 379.92,A -85,B 0,C 180,E1 -14692.277,E2 -14692.277} C_VEL
LIN {X 0,Y 333.739,Z 379.912,A -85,B 0,C 180,E1 -14696.245,E2 -14696.245} C_VEL
LIN {X 0,Y 333.722,Z 379.911,A -85,B 0,C 180,E1 -14696.638,E2 -14696.638} C_VEL
LIN {X 0,Y 333.032,Z 379.999,A -85,B 0,C 180,E1 -14697.646,E2 -14697.646} C_VEL
LIN {X 0,Y 330.126,Z 380.36,A -85,B 0,C 180,E1 -14699.284,E2 -14699.284} C_VEL
LIN {X 0,Y 327.684,Z 380.668,A -85,B 0,C 180,E1 -14700.611,E2 -14700.611} C_VEL
LIN {X 0,Y 326.654,Z 380.793,A -85,B 0,C 180,E1 -14701.639,E2 -14701.639} C_VEL
LIN {X 0,Y 326.581,Z 380.801,A -85,B 0,C 180,E1 -14701.987,E2 -14701.987} C_VEL
LIN {X 0,Y 326.613,Z 380.798,A -85,B 0,C 180,E1 -14705.519,E2 -14705.519} C_VEL
LIN {X 0,Y 326.611,Z 380.797,A -85,B 0,C 180,E1 -14709.226,E2 -14709.226} C_VEL
LIN {X 0,Y 326.585,Z 380.801,A -85,B 0,C 180,E1 -14712.973,E2 -14712.973} C_VEL
LIN {X 0,Y 326.629,Z 380.793,A -85,B 0,C 180,E1 -14717.017,E2 -14717.017} C_VEL
LIN {X 0,Y 326.643,Z 380.795,A -85,B 0,C 180,E1 -14720.764,E2 -14720.764} C_VEL
LIN {X 0,Y 326.61,Z 380.798,A -85,B 0,C 180,E1 -14724.479,E2 -14724.479} C_VEL
LIN {X 0,Y 326.604,Z 380.798,A -85,B 0,C 180,E1 -14727.454,E2 -14727.454} C_VEL
LIN {X 0,Y 326.643,Z 380.798,A -85,B 0,C 180,E1 -14730.339,E2 -14730.339} C_VEL
LIN {X 0,Y 326.685,Z 380.789,A -85,B 0,C 180,E1 -14734.515,E2 -14734.515} C_VEL
LIN {X 0,Y 326.648,Z 380.796,A -85,B 0,C 180,E1 -14738.545,E2 -14738.545} C_VEL
LIN {X 0,Y 326.739,Z 380.781,A -85,B 0,C 180,E1 -14741.177,E2 -14741.177} C_VEL
LIN {X 0,Y 326.757,Z 380.777,A -85,B 0,C 180,E1 -14745.433,E2 -14745.433} C_VEL
LIN {X 0,Y 326.767,Z 380.779,A -85,B 0,C 180,E1 -14748.838,E2 -14748.838} C_VEL
LIN {X 0,Y 326.972,Z 380.753,A -85,B 0,C 180,E1 -14752.59,E2 -14752.59} C_VEL
LIN {X 0,Y 326.772,Z 380.773,A -85,B 0,C 180,E1 -14755.064,E2 -14755.064} C_VEL
LIN {X 0,Y 327.041,Z 380.743,A -85,B 0,C 180,E1 -14757.536,E2 -14757.536} C_VEL
LIN {X 0,Y 327.211,Z 380.728,A -85,B 0,C 180,E1 -14760,E2 -14760} C_VEL
LIN {X 0,Y 327.042,Z 380.745,A -85,B 0,C 180,E1 -14762.463,E2 -14762.463} C_VEL
LIN {X 0,Y 326.989,Z 380.755,A -85,B 0,C 180,E1 -14766.169,E2 -14766.169} C_VEL
LIN {X 0,Y 326.908,Z 380.761,A -85,B 0,C 180,E1 -14768.655,E2 -14768.655} C_VEL
LIN {X 0,Y 326.732,Z 380.785,A -85,B 0,C 180,E1 -14772.421,E2 -14772.421} C_VEL
LIN {X 0,Y 326.747,Z 380.78,A -85,B 0,C 180,E1 -14774.958,E2 -14774.958} C_VEL
LIN {X 0,Y 326.729,Z 380.782,A -85,B 0,C 180,E1 -14778.84,E2 -14778.84} C_VEL
LIN {X 0,Y 326.615,Z 380.797,A -85,B 0,C 180,E1 -14782.788,E2 -14782.788} C_VEL
LIN {X 0,Y 326.684,Z 380.79,A -85,B 0,C 180,E1 -14785.484,E2 -14785.484} C_VEL
LIN {X 0,Y 326.642,Z 380.797,A -85,B 0,C 180,E1 -14789.661,E2 -14789.661} C_VEL
LIN {X 0,Y 326.601,Z 380.804,A -85,B 0,C 180,E1 -14794.02,E2 -14794.02} C_VEL
LIN {X 0,Y 326.624,Z 380.797,A -85,B 0,C 180,E1 -14797.24,E2 -14797.24} C_VEL
LIN {X 0,Y 326.631,Z 380.798,A -85,B 0,C 180,E1 -14800.203,E2 -14800.203} C_VEL
LIN {X 0,Y 326.622,Z 380.799,A -85,B 0,C 180,E1 -14803.516,E2 -14803.516} C_VEL
LIN {X 0,Y 326.594,Z 380.8,A -85,B 0,C 180,E1 -14807.025,E2 -14807.025} C_VEL
LIN {X 0,Y 326.609,Z 380.799,A -85,B 0,C 180,E1 -14810.773,E2 -14810.773} C_VEL
LIN {X 0,Y 326.61,Z 380.8,A -85,B 0,C 180,E1 -14814.481,E2 -14814.481} C_VEL
LIN {X 0,Y 326.672,Z 380.923,A -85,B 0,C 180,E1 -14818.463,E2 -14818.463} C_VEL
LIN {X 0,Y 329.398,Z 393.774,A -85,B 0,C 180,E1 -14822.006,E2 -14822.006} C_VEL
LIN {X 0,Y 330.564,Z 400.629,A -85,B 0,C 180,E1 -14823.823,E2 -14823.823} C_VEL
LIN {X 0,Y 329.973,Z 407.301,A -85,B 0,C 180,E1 -14825.461,E2 -14825.461} C_VEL
LIN {X 0,Y 329.39,Z 412.314,A -85,B 0,C 180,E1 -14826.679,E2 -14826.679} C_VEL
LIN {X 0,Y 334.841,Z 452.902,A -85,B 0,C 180,E1 -14827.93,E2 -14827.93} C_VEL
LIN {X 0,Y 333.51,Z 521.399,A -85,B 0,C 180,E1 -14829.412,E2 -14829.412} C_VEL
LIN {X 0,Y 332.848,Z 534.582,A -85,B 0,C 180,E1 -14829.934,E2 -14829.934} C_VEL
LIN {X 0,Y 331.913,Z 547.284,A -85,B 0,C 180,E1 -14830.68,E2 -14830.68} C_VEL
LIN {X 0,Y 330.864,Z 558.558,A -85,B 0,C 180,E1 -14831.581,E2 -14831.581} C_VEL
LIN {X 0,Y 329.62,Z 570.249,A -85,B 0,C 180,E1 -14832.793,E2 -14832.793} C_VEL
LIN {X 0,Y 328.408,Z 581.461,A -85,B 0,C 180,E1 -14834.268,E2 -14834.268} C_VEL
LIN {X 0,Y 327.556,Z 590.249,A -85,B 0,C 180,E1 -14835.716,E2 -14835.716} C_VEL
LIN {X 0,Y 326.516,Z 599.377,A -85,B 0,C 180,E1 -14837.571,E2 -14837.571} C_VEL
LIN {X 0,Y 325.769,Z 606.727,A -85,B 0,C 180,E1 -14839.434,E2 -14839.434} C_VEL
LIN {X 0,Y 325.311,Z 612.606,A -85,B 0,C 180,E1 -14841.302,E2 -14841.302} C_VEL
LIN {X 0,Y 325.047,Z 617.223,A -85,B 0,C 180,E1 -14843.17,E2 -14843.17} C_VEL
LIN {X 0,Y 324.955,Z 620.726,A -85,B 0,C 180,E1 -14845.037,E2 -14845.037} C_VEL
LIN {X 0,Y 324.969,Z 622.475,A -85,B 0,C 180,E1 -14846.28,E2 -14846.28} C_VEL
LIN {X 0,Y 325.007,Z 624.728,A -85,B 0,C 180,E1 -14848.761,E2 -14848.761} C_VEL
LIN {X 0,Y 325.039,Z 625.253,A -85,B 0,C 180,E1 -14850,E2 -14850} C_VEL
LIN {X 0,Y 324.964,Z 625.335,A -85,B 0,C 180,E1 -14851.239,E2 -14851.239} C_VEL
LIN {X 0,Y 324.94,Z 624.332,A -85,B 0,C 180,E1 -14853.72,E2 -14853.72} C_VEL
LIN {X 0,Y 324.919,Z 622.324,A -85,B 0,C 180,E1 -14855.744,E2 -14855.744} C_VEL
LIN {X 0,Y 325.244,Z 618.635,A -85,B 0,C 180,E1 -14858.074,E2 -14858.074} C_VEL
LIN {X 0,Y 325.723,Z 614.519,A -85,B 0,C 180,E1 -14859.94,E2 -14859.94} C_VEL
LIN {X 0,Y 326.602,Z 608.241,A -85,B 0,C 180,E1 -14862.111,E2 -14862.111} C_VEL
LIN {X 0,Y 327.829,Z 601.436,A -85,B 0,C 180,E1 -14863.956,E2 -14863.956} C_VEL
LIN {X 0,Y 329.159,Z 593.002,A -85,B 0,C 180,E1 -14865.797,E2 -14865.797} C_VEL
LIN {X 0,Y 330.527,Z 584.346,A -85,B 0,C 180,E1 -14867.318,E2 -14867.318} C_VEL
LIN {X 0,Y 332.292,Z 573.714,A -85,B 0,C 180,E1 -14868.816,E2 -14868.816} C_VEL
LIN {X 0,Y 333.869,Z 563.174,A -85,B 0,C 180,E1 -14870.002,E2 -14870.002} C_VEL
LIN {X 0,Y 335.386,Z 551.48,A -85,B 0,C 180,E1 -14871.029,E2 -14871.029} C_VEL
LIN {X 0,Y 336.741,Z 539.347,A -85,B 0,C 180,E1 -14871.824,E2 -14871.824} C_VEL
LIN {X 0,Y 337.768,Z 526.141,A -85,B 0,C 180,E1 -14872.437,E2 -14872.437} C_VEL
LIN {X 0,Y 338.359,Z 513.204,A -85,B 0,C 180,E1 -14872.799,E2 -14872.799} C_VEL
LIN {X 0,Y 339.655,Z 453.645,A -85,B 0,C 180,E1 -14874.075,E2 -14874.075} C_VEL
LIN {X 0,Y 336.169,Z 432.499,A -85,B 0,C 180,E1 -14874.879,E2 -14874.879} C_VEL
LIN {X 0,Y 331.934,Z 411.729,A -85,B 0,C 180,E1 -14875.775,E2 -14875.775} C_VEL
LIN {X 0,Y 332.548,Z 407.532,A -85,B 0,C 180,E1 -14876.833,E2 -14876.833} C_VEL
LIN {X 0,Y 331,Z 399.146,A -85,B 0,C 180,E1 -14879.231,E2 -14879.231} C_VEL
LIN {X 0,Y 328.38,Z 387.831,A -85,B 0,C 180,E1 -14882.663,E2 -14882.663} C_VEL
LIN {X 0,Y 326.63,Z 380.801,A -85,B 0,C 180,E1 -14884.973,E2 -14884.973} C_VEL
LIN {X 0,Y 326.621,Z 380.798,A -85,B 0,C 180,E1 -14888.608,E2 -14888.608} C_VEL
LIN {X 0,Y 326.574,Z 380.803,A -85,B 0,C 180,E1 -14891.845,E2 -14891.845} C_VEL
LIN {X 0,Y 326.594,Z 380.798,A -85,B 0,C 180,E1 -14895.244,E2 -14895.244} C_VEL
LIN {X 0,Y 326.625,Z 380.793,A -85,B 0,C 180,E1 -14898.858,E2 -14898.858} C_VEL
LIN {X 0,Y 326.642,Z 380.794,A -85,B 0,C 180,E1 -14901.394,E2 -14901.394} C_VEL
LIN {X 0,Y 326.614,Z 380.797,A -85,B 0,C 180,E1 -14904.851,E2 -14904.851} C_VEL
LIN {X 0,Y 326.602,Z 380.802,A -85,B 0,C 180,E1 -14907.455,E2 -14907.455} C_VEL
LIN {X 0,Y 326.655,Z 380.792,A -85,B 0,C 180,E1 -14910.341,E2 -14910.341} C_VEL
LIN {X 0,Y 326.684,Z 380.768,A -85,B 0,C 180,E1 -14914.516,E2 -14914.516} C_VEL
LIN {X 0,Y 326.64,Z 380.796,A -85,B 0,C 180,E1 -14918.545,E2 -14918.545} C_VEL
LIN {X 0,Y 326.738,Z 380.779,A -85,B 0,C 180,E1 -14921.177,E2 -14921.177} C_VEL
LIN {X 0,Y 326.756,Z 380.777,A -85,B 0,C 180,E1 -14925.433,E2 -14925.433} C_VEL
LIN {X 0,Y 326.766,Z 380.777,A -85,B 0,C 180,E1 -14928.839,E2 -14928.839} C_VEL
LIN {X 0,Y 326.972,Z 380.756,A -85,B 0,C 180,E1 -14932.59,E2 -14932.59} C_VEL
LIN {X 0,Y 326.773,Z 380.776,A -85,B 0,C 180,E1 -14935.065,E2 -14935.065} C_VEL
LIN {X 0,Y 327.041,Z 380.743,A -85,B 0,C 180,E1 -14937.537,E2 -14937.537} C_VEL
LIN {X 0,Y 327.211,Z 380.722,A -85,B 0,C 180,E1 -14940,E2 -14940} C_VEL
LIN {X 0,Y 327.041,Z 380.745,A -85,B 0,C 180,E1 -14942.464,E2 -14942.464} C_VEL
LIN {X 0,Y 326.952,Z 380.753,A -85,B 0,C 180,E1 -14946.665,E2 -14946.665} C_VEL
LIN {X 0,Y 326.799,Z 380.775,A -85,B 0,C 180,E1 -14949.907,E2 -14949.907} C_VEL
LIN {X 0,Y 326.753,Z 380.779,A -85,B 0,C 180,E1 -14953.686,E2 -14953.686} C_VEL
LIN {X 0,Y 326.693,Z 380.785,A -85,B 0,C 180,E1 -14957.529,E2 -14957.529} C_VEL
LIN {X 0,Y 326.659,Z 380.793,A -85,B 0,C 180,E1 -14960.136,E2 -14960.136} C_VEL
LIN {X 0,Y 326.647,Z 380.792,A -85,B 0,C 180,E1 -14964.13,E2 -14964.13} C_VEL
LIN {X 0,Y 326.68,Z 380.771,A -85,B 0,C 180,E1 -14966.859,E2 -14966.859} C_VEL
LIN {X 0,Y 326.635,Z 380.794,A -85,B 0,C 180,E1 -14970.612,E2 -14970.612} C_VEL
LIN {X 0,Y 326.603,Z 380.8,A -85,B 0,C 180,E1 -14974.02,E2 -14974.02} C_VEL
LIN {X 0,Y 326.626,Z 380.798,A -85,B 0,C 180,E1 -14977.24,E2 -14977.24} C_VEL
LIN {X 0,Y 326.633,Z 380.804,A -85,B 0,C 180,E1 -14980.204,E2 -14980.204} C_VEL
LIN {X 0,Y 326.627,Z 380.799,A -85,B 0,C 180,E1 -14983.515,E2 -14983.515} C_VEL
LIN {X 0,Y 326.616,Z 380.802,A -85,B 0,C 180,E1 -14987.021,E2 -14987.021} C_VEL
LIN {X 0,Y 326.644,Z 380.799,A -85,B 0,C 180,E1 -14991.395,E2 -14991.395} C_VEL
LIN {X 0,Y 326.661,Z 380.925,A -85,B 0,C 180,E1 -14993.199,E2 -14993.199} C_VEL
LIN {X 0,Y 327.82,Z 385.67,A -85,B 0,C 180,E1 -14994.883,E2 -14994.883} C_VEL
LIN {X 0,Y 337.705,Z 407.263,A -85,B 0,C 180,E1 -14996.352,E2 -14996.352} C_VEL
LIN {X 0,Y 340.657,Z 414.624,A -85,B 0,C 180,E1 -14996.791,E2 -14996.791} C_VEL
LIN {X 0,Y 338.645,Z 492.153,A -85,B 0,C 180,E1 -14998.465,E2 -14998.465} C_VEL
LIN {X 0,Y 337.996,Z 504.305,A -85,B 0,C 180,E1 -14998.941,E2 -14998.941} C_VEL
LIN {X 0,Y 336.967,Z 517.427,A -85,B 0,C 180,E1 -14999.705,E2 -14999.705} C_VEL
LIN {X 0,Y 335.766,Z 528.098,A -85,B 0,C 180,E1 -15000.536,E2 -15000.536} C_VEL
LIN {X 0,Y 334.506,Z 539.609,A -85,B 0,C 180,E1 -15001.721,E2 -15001.721} C_VEL
LIN {X 0,Y 332.823,Z 550.816,A -85,B 0,C 180,E1 -15003.17,E2 -15003.17} C_VEL
LIN {X 0,Y 331.443,Z 559.504,A -85,B 0,C 180,E1 -15004.572,E2 -15004.572} C_VEL
LIN {X 0,Y 329.892,Z 568.433,A -85,B 0,C 180,E1 -15006.36,E2 -15006.36} C_VEL
LIN {X 0,Y 328.415,Z 576.282,A -85,B 0,C 180,E1 -15008.338,E2 -15008.338} C_VEL
LIN {X 0,Y 327.483,Z 581.297,A -85,B 0,C 180,E1 -15009.918,E2 -15009.918} C_VEL
LIN {X 0,Y 326.618,Z 586.127,A -85,B 0,C 180,E1 -15011.82,E2 -15011.82} C_VEL
LIN {X 0,Y 325.946,Z 589.799,A -85,B 0,C 180,E1 -15013.722,E2 -15013.722} C_VEL
LIN {X 0,Y 325.622,Z 591.68,A -85,B 0,C 180,E1 -15014.99,E2 -15014.99} C_VEL
LIN {X 0,Y 325.38,Z 593.213,A -85,B 0,C 180,E1 -15016.405,E2 -15016.405} C_VEL
LIN {X 0,Y 325.005,Z 594.664,A -85,B 0,C 180,E1 -15018.778,E2 -15018.778} C_VEL
LIN {X 0,Y 324.897,Z 594.863,A -85,B 0,C 180,E1 -15020.035,E2 -15020.035} C_VEL
LIN {X 0,Y 324.921,Z 594.622,A -85,B 0,C 180,E1 -15021.292,E2 -15021.292} C_VEL
LIN {X 0,Y 324.986,Z 593.991,A -85,B 0,C 180,E1 -15022.545,E2 -15022.545} C_VEL
LIN {X 0,Y 325.101,Z 592.831,A -85,B 0,C 180,E1 -15023.952,E2 -15023.952} C_VEL
LIN {X 0,Y 325.23,Z 589.687,A -85,B 0,C 180,E1 -15026.283,E2 -15026.283} C_VEL
LIN {X 0,Y 325.598,Z 586.061,A -85,B 0,C 180,E1 -15028.145,E2 -15028.145} C_VEL
LIN {X 0,Y 325.959,Z 581.347,A -85,B 0,C 180,E1 -15030,E2 -15030} C_VEL
LIN {X 0,Y 326.839,Z 574.263,A -85,B 0,C 180,E1 -15032.157,E2 -15032.157} C_VEL
LIN {X 0,Y 327.795,Z 566.551,A -85,B 0,C 180,E1 -15033.996,E2 -15033.996} C_VEL
LIN {X 0,Y 328.816,Z 556.929,A -85,B 0,C 180,E1 -15035.827,E2 -15035.827} C_VEL
LIN {X 0,Y 330.021,Z 546.954,A -85,B 0,C 180,E1 -15037.341,E2 -15037.341} C_VEL
LIN {X 0,Y 331.162,Z 535.67,A -85,B 0,C 180,E1 -15038.697,E2 -15038.697} C_VEL
LIN {X 0,Y 332.067,Z 524.638,A -85,B 0,C 180,E1 -15039.748,E2 -15039.748} C_VEL
LIN {X 0,Y 332.934,Z 512.345,A -85,B 0,C 180,E1 -15040.644,E2 -15040.644} C_VEL
LIN {X 0,Y 333.574,Z 499.265,A -85,B 0,C 180,E1 -15041.315,E2 -15041.315} C_VEL
LIN {X 0,Y 333.946,Z 486.683,A -85,B 0,C 180,E1 -15041.725,E2 -15041.725} C_VEL
LIN {X 0,Y 335.436,Z 410.348,A -85,B 0,C 180,E1 -15043.346,E2 -15043.346} C_VEL
LIN {X 0,Y 333.55,Z 402.171,A -85,B 0,C 180,E1 -15043.644,E2 -15043.644} C_VEL
LIN {X 0,Y 327.519,Z 384.635,A -85,B 0,C 180,E1 -15044.448,E2 -15044.448} C_VEL
LIN {X 0,Y 326.768,Z 380.784,A -85,B 0,C 180,E1 -15045.755,E2 -15045.755} C_VEL
LIN {X 0,Y 326.738,Z 380.785,A -85,B 0,C 180,E1 -15048.838,E2 -15048.838} C_VEL
LIN {X 0,Y 326.624,Z 380.799,A -85,B 0,C 180,E1 -15052.787,E2 -15052.787} C_VEL
LIN {X 0,Y 326.677,Z 380.789,A -85,B 0,C 180,E1 -15056.648,E2 -15056.648} C_VEL
LIN {X 0,Y 326.663,Z 380.791,A -85,B 0,C 180,E1 -15059.658,E2 -15059.658} C_VEL
LIN {X 0,Y 326.581,Z 380.801,A -85,B 0,C 180,E1 -15061.987,E2 -15061.987} C_VEL
LIN {X 0,Y 325.932,Z 380.886,A -85,B 0,C 180,E1 -15063.017,E2 -15063.017} C_VEL
LIN {X 0,Y 323.064,Z 381.243,A -85,B 0,C 180,E1 -15064.694,E2 -15064.694} C_VEL
LIN {X 0,Y 320.637,Z 381.545,A -85,B 0,C 180,E1 -15066.053,E2 -15066.053} C_VEL
LIN {X 0,Y 319.62,Z 381.669,A -85,B 0,C 180,E1 -15067.105,E2 -15067.105} C_VEL
LIN {X 0,Y 319.552,Z 381.677,A -85,B 0,C 180,E1 -15067.461,E2 -15067.461} C_VEL
LIN {X 0,Y 319.528,Z 381.678,A -85,B 0,C 180,E1 -15071.287,E2 -15071.287} C_VEL
LIN {X 0,Y 319.566,Z 381.677,A -85,B 0,C 180,E1 -15074.728,E2 -15074.728} C_VEL
LIN {X 0,Y 319.595,Z 381.675,A -85,B 0,C 180,E1 -15078.388,E2 -15078.388} C_VEL
LIN {X 0,Y 319.598,Z 381.674,A -85,B 0,C 180,E1 -15081.995,E2 -15081.995} C_VEL
LIN {X 0,Y 319.557,Z 381.672,A -85,B 0,C 180,E1 -15085.122,E2 -15085.122} C_VEL
LIN {X 0,Y 319.562,Z 381.676,A -85,B 0,C 180,E1 -15089.058,E2 -15089.058} C_VEL
LIN {X 0,Y 319.601,Z 381.672,A -85,B 0,C 180,E1 -15092.497,E2 -15092.497} C_VEL
LIN {X 0,Y 319.6,Z 381.668,A -85,B 0,C 180,E1 -15095.303,E2 -15095.303} C_VEL
LIN {X 0,Y 319.617,Z 381.669,A -85,B 0,C 180,E1 -15099.401,E2 -15099.401} C_VEL
LIN {X 0,Y 319.653,Z 381.668,A -85,B 0,C 180,E1 -15102.072,E2 -15102.072} C_VEL
LIN {X 0,Y 319.727,Z 381.655,A -85,B 0,C 180,E1 -15106.007,E2 -15106.007} C_VEL
LIN {X 0,Y 319.753,Z 381.655,A -85,B 0,C 180,E1 -15109.872,E2 -15109.872} C_VEL
LIN {X 0,Y 319.926,Z 381.631,A -85,B 0,C 180,E1 -15112.426,E2 -15112.426} C_VEL
LIN {X 0,Y 319.742,Z 381.648,A -85,B 0,C 180,E1 -15114.956,E2 -15114.956} C_VEL
LIN {X 0,Y 319.985,Z 381.622,A -85,B 0,C 180,E1 -15117.482,E2 -15117.482} C_VEL
LIN {X 0,Y 320.162,Z 381.605,A -85,B 0,C 180,E1 -15120,E2 -15120} C_VEL
LIN {X 0,Y 319.985,Z 381.624,A -85,B 0,C 180,E1 -15122.517,E2 -15122.517} C_VEL
LIN {X 0,Y 319.945,Z 381.631,A -85,B 0,C 180,E1 -15126.305,E2 -15126.305} C_VEL
LIN {X 0,Y 319.836,Z 381.641,A -85,B 0,C 180,E1 -15128.848,E2 -15128.848} C_VEL
LIN {X 0,Y 319.678,Z 381.661,A -85,B 0,C 180,E1 -15132.7,E2 -15132.7} C_VEL
LIN {X 0,Y 319.693,Z 381.66,A -85,B 0,C 180,E1 -15135.296,E2 -15135.296} C_VEL
LIN {X 0,Y 319.671,Z 381.662,A -85,B 0,C 180,E1 -15139.255,E2 -15139.255} C_VEL
LIN {X 0,Y 319.564,Z 381.676,A -85,B 0,C 180,E1 -15143.32,E2 -15143.32} C_VEL
LIN {X 0,Y 319.628,Z 381.673,A -85,B 0,C 180,E1 -15146.088,E2 -15146.088} C_VEL
LIN {X 0,Y 319.573,Z 381.674,A -85,B 0,C 180,E1 -15148.935,E2 -15148.935} C_VEL
LIN {X 0,Y 319.525,Z 381.686,A -85,B 0,C 180,E1 -15151.862,E2 -15151.862} C_VEL
LIN {X 0,Y 319.575,Z 381.677,A -85,B 0,C 180,E1 -15155.544,E2 -15155.544} C_VEL
LIN {X 0,Y 319.595,Z 381.677,A -85,B 0,C 180,E1 -15158.005,E2 -15158.005} C_VEL
LIN {X 0,Y 319.593,Z 381.675,A -85,B 0,C 180,E1 -15161.612,E2 -15161.612} C_VEL
LIN {X 0,Y 319.567,Z 381.676,A -85,B 0,C 180,E1 -15165.273,E2 -15165.273} C_VEL
LIN {X 0,Y 319.53,Z 381.681,A -85,B 0,C 180,E1 -15168.713,E2 -15168.713} C_VEL
LIN {X 0,Y 319.575,Z 381.676,A -85,B 0,C 180,E1 -15172.345,E2 -15172.345} C_VEL
LIN {X 0,Y 319.559,Z 381.678,A -85,B 0,C 180,E1 -15175.124,E2 -15175.124} C_VEL
LIN {X 0,Y 319.608,Z 381.765,A -85,B 0,C 180,E1 -15178.101,E2 -15178.101} C_VEL
LIN {X 0,Y 322.049,Z 393.072,A -85,B 0,C 180,E1 -15181.309,E2 -15181.309} C_VEL
LIN {X 0,Y 323.564,Z 401.385,A -85,B 0,C 180,E1 -15183.579,E2 -15183.579} C_VEL
LIN {X 0,Y 323.18,Z 406.645,A -85,B 0,C 180,E1 -15184.91,E2 -15184.91} C_VEL
LIN {X 0,Y 322.535,Z 412.054,A -85,B 0,C 180,E1 -15186.246,E2 -15186.246} C_VEL
LIN {X 0,Y 328.107,Z 453.452,A -85,B 0,C 180,E1 -15187.547,E2 -15187.547} C_VEL
LIN {X 0,Y 326.842,Z 517.149,A -85,B 0,C 180,E1 -15188.931,E2 -15188.931} C_VEL
LIN {X 0,Y 326.336,Z 530.464,A -85,B 0,C 180,E1 -15189.392,E2 -15189.392} C_VEL
LIN {X 0,Y 325.377,Z 543.659,A -85,B 0,C 180,E1 -15190.112,E2 -15190.112} C_VEL
LIN {X 0,Y 324.282,Z 555.719,A -85,B 0,C 180,E1 -15191.03,E2 -15191.03} C_VEL
LIN {X 0,Y 323.122,Z 566.649,A -85,B 0,C 180,E1 -15192.108,E2 -15192.108} C_VEL
LIN {X 0,Y 321.962,Z 576.701,A -85,B 0,C 180,E1 -15193.352,E2 -15193.352} C_VEL
LIN {X 0,Y 321.052,Z 585.949,A -85,B 0,C 180,E1 -15194.771,E2 -15194.771} C_VEL
LIN {X 0,Y 320.034,Z 594.388,A -85,B 0,C 180,E1 -15196.346,E2 -15196.346} C_VEL
LIN {X 0,Y 319.1,Z 602.639,A -85,B 0,C 180,E1 -15198.245,E2 -15198.245} C_VEL
LIN {X 0,Y 318.554,Z 608.255,A -85,B 0,C 180,E1 -15199.834,E2 -15199.834} C_VEL
LIN {X 0,Y 318.146,Z 613.739,A -85,B 0,C 180,E1 -15201.745,E2 -15201.745} C_VEL
LIN {X 0,Y 317.915,Z 618.014,A -85,B 0,C 180,E1 -15203.654,E2 -15203.654} C_VEL
LIN {X 0,Y 317.868,Z 620.279,A -85,B 0,C 180,E1 -15204.926,E2 -15204.926} C_VEL
LIN {X 0,Y 317.895,Z 622.062,A -85,B 0,C 180,E1 -15206.197,E2 -15206.197} C_VEL
LIN {X 0,Y 317.911,Z 624.35,A -85,B 0,C 180,E1 -15208.733,E2 -15208.733} C_VEL
LIN {X 0,Y 317.948,Z 624.9,A -85,B 0,C 180,E1 -15210,E2 -15210} C_VEL
LIN {X 0,Y 317.868,Z 625.009,A -85,B 0,C 180,E1 -15211.267,E2 -15211.267} C_VEL
LIN {X 0,Y 317.843,Z 624.041,A -85,B 0,C 180,E1 -15213.803,E2 -15213.803} C_VEL
LIN {X 0,Y 317.838,Z 622.257,A -85,B 0,C 180,E1 -15215.711,E2 -15215.711} C_VEL
LIN {X 0,Y 318.193,Z 618.437,A -85,B 0,C 180,E1 -15218.254,E2 -15218.254} C_VEL
LIN {X 0,Y 318.685,Z 614.36,A -85,B 0,C 180,E1 -15220.161,E2 -15220.161} C_VEL
LIN {X 0,Y 319.619,Z 608.128,A -85,B 0,C 180,E1 -15222.379,E2 -15222.379} C_VEL
LIN {X 0,Y 320.937,Z 601.374,A -85,B 0,C 180,E1 -15224.262,E2 -15224.262} C_VEL
LIN {X 0,Y 322.216,Z 593.589,A -85,B 0,C 180,E1 -15226.023,E2 -15226.023} C_VEL
LIN {X 0,Y 323.737,Z 584.444,A -85,B 0,C 180,E1 -15227.693,E2 -15227.693} C_VEL
LIN {X 0,Y 325.602,Z 573.899,A -85,B 0,C 180,E1 -15229.218,E2 -15229.218} C_VEL
LIN {X 0,Y 327.223,Z 563.472,A -85,B 0,C 180,E1 -15230.426,E2 -15230.426} C_VEL
LIN {X 0,Y 328.801,Z 552.021,A -85,B 0,C 180,E1 -15231.471,E2 -15231.471} C_VEL
LIN {X 0,Y 330.315,Z 538.886,A -85,B 0,C 180,E1 -15232.353,E2 -15232.353} C_VEL
LIN {X 0,Y 331.396,Z 525.632,A -85,B 0,C 180,E1 -15232.975,E2 -15232.975} C_VEL
LIN {X 0,Y 332.011,Z 512.546,A -85,B 0,C 180,E1 -15233.343,E2 -15233.343} C_VEL
LIN {X 0,Y 333.343,Z 454.763,A -85,B 0,C 180,E1 -15234.602,E2 -15234.602} C_VEL
LIN {X 0,Y 330.006,Z 434.175,A -85,B 0,C 180,E1 -15235.405,E2 -15235.405} C_VEL
LIN {X 0,Y 325.775,Z 413.557,A -85,B 0,C 180,E1 -15236.319,E2 -15236.319} C_VEL
LIN {X 0,Y 325.394,Z 411.211,A -85,B 0,C 180,E1 -15236.462,E2 -15236.462} C_VEL
LIN {X 0,Y 325.651,Z 409.333,A -85,B 0,C 180,E1 -15236.949,E2 -15236.949} C_VEL
LIN {X 0,Y 324.341,Z 401.745,A -85,B 0,C 180,E1 -15239.158,E2 -15239.158} C_VEL
LIN {X 0,Y 321.715,Z 390.222,A -85,B 0,C 180,E1 -15242.728,E2 -15242.728} C_VEL
LIN {X 0,Y 319.58,Z 381.678,A -85,B 0,C 180,E1 -15245.612,E2 -15245.612} C_VEL
LIN {X 0,Y 319.57,Z 381.679,A -85,B 0,C 180,E1 -15248.007,E2 -15248.007} C_VEL
LIN {X 0,Y 319.523,Z 381.682,A -85,B 0,C 180,E1 -15251.596,E2 -15251.596} C_VEL
LIN {X 0,Y 319.573,Z 381.673,A -85,B 0,C 180,E1 -15255.272,E2 -15255.272} C_VEL
LIN {X 0,Y 319.576,Z 381.671,A -85,B 0,C 180,E1 -15258.719,E2 -15258.719} C_VEL
LIN {X 0,Y 319.593,Z 381.67,A -85,B 0,C 180,E1 -15262.339,E2 -15262.339} C_VEL
LIN {X 0,Y 319.555,Z 381.678,A -85,B 0,C 180,E1 -15265.123,E2 -15265.123} C_VEL
LIN {X 0,Y 319.565,Z 381.678,A -85,B 0,C 180,E1 -15269.058,E2 -15269.058} C_VEL
LIN {X 0,Y 319.603,Z 381.671,A -85,B 0,C 180,E1 -15272.498,E2 -15272.498} C_VEL
LIN {X 0,Y 319.598,Z 381.648,A -85,B 0,C 180,E1 -15275.304,E2 -15275.304} C_VEL
LIN {X 0,Y 319.591,Z 381.674,A -85,B 0,C 180,E1 -15278.048,E2 -15278.048} C_VEL
LIN {X 0,Y 319.683,Z 381.657,A -85,B 0,C 180,E1 -15280.962,E2 -15280.962} C_VEL
LIN {X 0,Y 319.724,Z 381.652,A -85,B 0,C 180,E1 -15285.276,E2 -15285.276} C_VEL
LIN {X 0,Y 319.753,Z 381.648,A -85,B 0,C 180,E1 -15289.873,E2 -15289.873} C_VEL
LIN {X 0,Y 319.926,Z 381.633,A -85,B 0,C 180,E1 -15292.426,E2 -15292.426} C_VEL
LIN {X 0,Y 319.742,Z 381.65,A -85,B 0,C 180,E1 -15294.956,E2 -15294.956} C_VEL
LIN {X 0,Y 319.985,Z 381.622,A -85,B 0,C 180,E1 -15297.483,E2 -15297.483} C_VEL
LIN {X 0,Y 320.162,Z 381.6,A -85,B 0,C 180,E1 -15300,E2 -15300} C_VEL
LIN {X 0,Y 319.985,Z 381.623,A -85,B 0,C 180,E1 -15302.518,E2 -15302.518} C_VEL
LIN {X 0,Y 319.913,Z 381.632,A -85,B 0,C 180,E1 -15306.654,E2 -15306.654} C_VEL
LIN {X 0,Y 319.746,Z 381.655,A -85,B 0,C 180,E1 -15310.128,E2 -15310.128} C_VEL
LIN {X 0,Y 319.725,Z 381.661,A -85,B 0,C 180,E1 -15314.725,E2 -15314.725} C_VEL
LIN {X 0,Y 319.684,Z 381.663,A -85,B 0,C 180,E1 -15319.039,E2 -15319.039} C_VEL
LIN {X 0,Y 319.565,Z 381.677,A -85,B 0,C 180,E1 -15323.32,E2 -15323.32} C_VEL
LIN {X 0,Y 319.614,Z 381.65,A -85,B 0,C 180,E1 -15326.09,E2 -15326.09} C_VEL
LIN {X 0,Y 319.586,Z 381.675,A -85,B 0,C 180,E1 -15328.935,E2 -15328.935} C_VEL
LIN {X 0,Y 319.528,Z 381.679,A -85,B 0,C 180,E1 -15331.863,E2 -15331.863} C_VEL
LIN {X 0,Y 319.577,Z 381.678,A -85,B 0,C 180,E1 -15335.544,E2 -15335.544} C_VEL
LIN {X 0,Y 319.597,Z 381.678,A -85,B 0,C 180,E1 -15338.005,E2 -15338.005} C_VEL
LIN {X 0,Y 319.595,Z 381.673,A -85,B 0,C 180,E1 -15341.612,E2 -15341.612} C_VEL
LIN {X 0,Y 319.58,Z 381.681,A -85,B 0,C 180,E1 -15345.275,E2 -15345.275} C_VEL
LIN {X 0,Y 319.546,Z 381.685,A -85,B 0,C 180,E1 -15348.716,E2 -15348.716} C_VEL
LIN {X 0,Y 319.595,Z 381.72,A -85,B 0,C 180,E1 -15352.58,E2 -15352.58} C_VEL
LIN {X 0,Y 320.602,Z 385.957,A -85,B 0,C 180,E1 -15354.147,E2 -15354.147} C_VEL
LIN {X 0,Y 329.595,Z 405.051,A -85,B 0,C 180,E1 -15355.536,E2 -15355.536} C_VEL
LIN {X 0,Y 334.314,Z 416.294,A -85,B 0,C 180,E1 -15356.255,E2 -15356.255} C_VEL
LIN {X 0,Y 332.281,Z 492.532,A -85,B 0,C 180,E1 -15357.934,E2 -15357.934} C_VEL
LIN {X 0,Y 331.564,Z 505.26,A -85,B 0,C 180,E1 -15358.448,E2 -15358.448} C_VEL
LIN {X 0,Y 330.489,Z 518.214,A -85,B 0,C 180,E1 -15359.224,E2 -15359.224} C_VEL
LIN {X 0,Y 329.243,Z 528.773,A -85,B 0,C 180,E1 -15360.07,E2 -15360.07} C_VEL
LIN {X 0,Y 327.965,Z 539.93,A -85,B 0,C 180,E1 -15361.245,E2 -15361.245} C_VEL
LIN {X 0,Y 326.334,Z 550.266,A -85,B 0,C 180,E1 -15362.592,E2 -15362.592} C_VEL
LIN {X 0,Y 324.864,Z 559.098,A -85,B 0,C 180,E1 -15364.019,E2 -15364.019} C_VEL
LIN {X 0,Y 323.449,Z 567.183,A -85,B 0,C 180,E1 -15365.617,E2 -15365.617} C_VEL
LIN {X 0,Y 321.917,Z 575.026,A -85,B 0,C 180,E1 -15367.54,E2 -15367.54} C_VEL
LIN {X 0,Y 320.654,Z 581.259,A -85,B 0,C 180,E1 -15369.471,E2 -15369.471} C_VEL
LIN {X 0,Y 319.688,Z 586.233,A -85,B 0,C 180,E1 -15371.441,E2 -15371.441} C_VEL
LIN {X 0,Y 318.975,Z 589.916,A -85,B 0,C 180,E1 -15373.356,E2 -15373.356} C_VEL
LIN {X 0,Y 318.634,Z 591.834,A -85,B 0,C 180,E1 -15374.652,E2 -15374.652} C_VEL
LIN {X 0,Y 318.302,Z 593.602,A -85,B 0,C 180,E1 -15376.292,E2 -15376.292} C_VEL
LIN {X 0,Y 317.937,Z 594.952,A -85,B 0,C 180,E1 -15378.525,E2 -15378.525} C_VEL
LIN {X 0,Y 317.815,Z 595.192,A -85,B 0,C 180,E1 -15379.811,E2 -15379.811} C_VEL
LIN {X 0,Y 317.821,Z 595.008,A -85,B 0,C 180,E1 -15381.096,E2 -15381.096} C_VEL
LIN {X 0,Y 317.899,Z 594.408,A -85,B 0,C 180,E1 -15382.378,E2 -15382.378} C_VEL
LIN {X 0,Y 318.03,Z 593.152,A -85,B 0,C 180,E1 -15383.959,E2 -15383.959} C_VEL
LIN {X 0,Y 318.141,Z 590.236,A -85,B 0,C 180,E1 -15386.2,E2 -15386.2} C_VEL
LIN {X 0,Y 318.515,Z 586.682,A -85,B 0,C 180,E1 -15388.103,E2 -15388.103} C_VEL
LIN {X 0,Y 318.889,Z 582.045,A -85,B 0,C 180,E1 -15390,E2 -15390} C_VEL
LIN {X 0,Y 319.761,Z 575.048,A -85,B 0,C 180,E1 -15392.204,E2 -15392.204} C_VEL
LIN {X 0,Y 320.73,Z 567.477,A -85,B 0,C 180,E1 -15394.084,E2 -15394.084} C_VEL
LIN {X 0,Y 321.796,Z 557.981,A -85,B 0,C 180,E1 -15395.954,E2 -15395.954} C_VEL
LIN {X 0,Y 323.018,Z 548.166,A -85,B 0,C 180,E1 -15397.501,E2 -15397.501} C_VEL
LIN {X 0,Y 324.214,Z 537.15,A -85,B 0,C 180,E1 -15398.885,E2 -15398.885} C_VEL
LIN {X 0,Y 325.272,Z 524.646,A -85,B 0,C 180,E1 -15400.111,E2 -15400.111} C_VEL
LIN {X 0,Y 326.114,Z 513.408,A -85,B 0,C 180,E1 -15400.948,E2 -15400.948} C_VEL
LIN {X 0,Y 326.771,Z 500.734,A -85,B 0,C 180,E1 -15401.632,E2 -15401.632} C_VEL
LIN {X 0,Y 327.19,Z 487.402,A -85,B 0,C 180,E1 -15402.089,E2 -15402.089} C_VEL
LIN {X 0,Y 328.724,Z 411.241,A -85,B 0,C 180,E1 -15403.739,E2 -15403.739} C_VEL
LIN {X 0,Y 326.818,Z 403.296,A -85,B 0,C 180,E1 -15404.042,E2 -15404.042} C_VEL
LIN {X 0,Y 320.34,Z 384.902,A -85,B 0,C 180,E1 -15404.935,E2 -15404.935} C_VEL
LIN {X 0,Y 319.711,Z 381.663,A -85,B 0,C 180,E1 -15406.03,E2 -15406.03} C_VEL
LIN {X 0,Y 319.679,Z 381.663,A -85,B 0,C 180,E1 -15409.254,E2 -15409.254} C_VEL
LIN {X 0,Y 319.573,Z 381.675,A -85,B 0,C 180,E1 -15413.319,E2 -15413.319} C_VEL
LIN {X 0,Y 319.638,Z 381.666,A -85,B 0,C 180,E1 -15416.087,E2 -15416.087} C_VEL
LIN {X 0,Y 319.6,Z 381.672,A -85,B 0,C 180,E1 -15418.932,E2 -15418.932} C_VEL
LIN {X 0,Y 319.531,Z 381.68,A -85,B 0,C 180,E1 -15421.981,E2 -15421.981} C_VEL
LIN {X 0,Y 319.58,Z 381.674,A -85,B 0,C 180,E1 -15425.542,E2 -15425.542} C_VEL
LIN {X 0,Y 319.552,Z 381.677,A -85,B 0,C 180,E1 -15427.461,E2 -15427.461} C_VEL
LIN {X 0,Y 318.92,Z 381.76,A -85,B 0,C 180,E1 -15428.513,E2 -15428.513} C_VEL
LIN {X 0,Y 316.066,Z 382.116,A -85,B 0,C 180,E1 -15430.224,E2 -15430.224} C_VEL
LIN {X 0,Y 313.623,Z 382.419,A -85,B 0,C 180,E1 -15431.611,E2 -15431.611} C_VEL
LIN {X 0,Y 312.572,Z 382.549,A -85,B 0,C 180,E1 -15432.685,E2 -15432.685} C_VEL
LIN {X 0,Y 312.486,Z 382.557,A -85,B 0,C 180,E1 -15433.049,E2 -15433.049} C_VEL
LIN {X 0,Y 312.537,Z 382.553,A -85,B 0,C 180,E1 -15436.019,E2 -15436.019} C_VEL
LIN {X 0,Y 312.545,Z 382.551,A -85,B 0,C 180,E1 -15439.864,E2 -15439.864} C_VEL
LIN {X 0,Y 312.551,Z 382.55,A -85,B 0,C 180,E1 -15442.618,E2 -15442.618} C_VEL
LIN {X 0,Y 312.516,Z 382.555,A -85,B 0,C 180,E1 -15446.31,E2 -15446.31} C_VEL
LIN {X 0,Y 312.534,Z 382.556,A -85,B 0,C 180,E1 -15450.348,E2 -15450.348} C_VEL
LIN {X 0,Y 312.598,Z 382.544,A -85,B 0,C 180,E1 -15454.064,E2 -15454.064} C_VEL
LIN {X 0,Y 312.583,Z 382.545,A -85,B 0,C 180,E1 -15457.528,E2 -15457.528} C_VEL
LIN {X 0,Y 312.633,Z 382.539,A -85,B 0,C 180,E1 -15461.656,E2 -15461.656} C_VEL
LIN {X 0,Y 312.688,Z 382.529,A -85,B 0,C 180,E1 -15465.686,E2 -15465.686} C_VEL
LIN {X 0,Y 312.698,Z 382.532,A -85,B 0,C 180,E1 -15469.641,E2 -15469.641} C_VEL
LIN {X 0,Y 312.865,Z 382.512,A -85,B 0,C 180,E1 -15472.254,E2 -15472.254} C_VEL
LIN {X 0,Y 312.712,Z 382.523,A -85,B 0,C 180,E1 -15474.842,E2 -15474.842} C_VEL
LIN {X 0,Y 312.986,Z 382.495,A -85,B 0,C 180,E1 -15478.713,E2 -15478.713} C_VEL
LIN {X 0,Y 313.114,Z 382.483,A -85,B 0,C 180,E1 -15480,E2 -15480} C_VEL
LIN {X 0,Y 312.932,Z 382.502,A -85,B 0,C 180,E1 -15482.574,E2 -15482.574} C_VEL
LIN {X 0,Y 312.903,Z 382.507,A -85,B 0,C 180,E1 -15486.448,E2 -15486.448} C_VEL
LIN {X 0,Y 312.781,Z 382.52,A -85,B 0,C 180,E1 -15489.049,E2 -15489.049} C_VEL
LIN {X 0,Y 312.63,Z 382.539,A -85,B 0,C 180,E1 -15492.991,E2 -15492.991} C_VEL
LIN {X 0,Y 312.632,Z 382.541,A -85,B 0,C 180,E1 -15495.65,E2 -15495.65} C_VEL
LIN {X 0,Y 312.601,Z 382.545,A -85,B 0,C 180,E1 -15499.708,E2 -15499.708} C_VEL
LIN {X 0,Y 312.54,Z 382.55,A -85,B 0,C 180,E1 -15502.79,E2 -15502.79} C_VEL
LIN {X 0,Y 312.596,Z 382.549,A -85,B 0,C 180,E1 -15505.936,E2 -15505.936} C_VEL
LIN {X 0,Y 312.532,Z 382.555,A -85,B 0,C 180,E1 -15509.651,E2 -15509.651} C_VEL
LIN {X 0,Y 312.514,Z 382.558,A -85,B 0,C 180,E1 -15513.689,E2 -15513.689} C_VEL
LIN {X 0,Y 312.548,Z 382.551,A -85,B 0,C 180,E1 -15517.382,E2 -15517.382} C_VEL
LIN {X 0,Y 312.529,Z 382.553,A -85,B 0,C 180,E1 -15520.703,E2 -15520.703} C_VEL
LIN {X 0,Y 312.53,Z 382.554,A -85,B 0,C 180,E1 -15524.195,E2 -15524.195} C_VEL
LIN {X 0,Y 312.519,Z 382.559,A -85,B 0,C 180,E1 -15527.912,E2 -15527.912} C_VEL
LIN {X 0,Y 312.532,Z 382.557,A -85,B 0,C 180,E1 -15531.911,E2 -15531.911} C_VEL
LIN {X 0,Y 312.505,Z 382.56,A -85,B 0,C 180,E1 -15535.791,E2 -15535.791} C_VEL
LIN {X 0,Y 312.574,Z 382.736,A -85,B 0,C 180,E1 -15537.76,E2 -15537.76} C_VEL
LIN {X 0,Y 314.813,Z 393.148,A -85,B 0,C 180,E1 -15540.795,E2 -15540.795} C_VEL
LIN {X 0,Y 316.451,Z 401.739,A -85,B 0,C 180,E1 -15543.208,E2 -15543.208} C_VEL
LIN {X 0,Y 316.608,Z 404.691,A -85,B 0,C 180,E1 -15543.998,E2 -15543.998} C_VEL
LIN {X 0,Y 315.727,Z 411.626,A -85,B 0,C 180,E1 -15545.765,E2 -15545.765} C_VEL
LIN {X 0,Y 321.314,Z 453.326,A -85,B 0,C 180,E1 -15547.129,E2 -15547.129} C_VEL
LIN {X 0,Y 320.155,Z 514.035,A -85,B 0,C 180,E1 -15548.469,E2 -15548.469} C_VEL
LIN {X 0,Y 319.748,Z 527.571,A -85,B 0,C 180,E1 -15548.905,E2 -15548.905} C_VEL
LIN {X 0,Y 318.762,Z 541.089,A -85,B 0,C 180,E1 -15549.597,E2 -15549.597} C_VEL
LIN {X 0,Y 317.743,Z 552.813,A -85,B 0,C 180,E1 -15550.456,E2 -15550.456} C_VEL
LIN {X 0,Y 316.482,Z 564.232,A -85,B 0,C 180,E1 -15551.552,E2 -15551.552} C_VEL
LIN {X 0,Y 315.089,Z 575.843,A -85,B 0,C 180,E1 -15552.978,E2 -15552.978} C_VEL
LIN {X 0,Y 314.125,Z 585.206,A -85,B 0,C 180,E1 -15554.427,E2 -15554.427} C_VEL
LIN {X 0,Y 313.059,Z 593.716,A -85,B 0,C 180,E1 -15556.035,E2 -15556.035} C_VEL
LIN {X 0,Y 312.089,Z 602.026,A -85,B 0,C 180,E1 -15557.977,E2 -15557.977} C_VEL
LIN {X 0,Y 311.424,Z 608.714,A -85,B 0,C 180,E1 -15559.928,E2 -15559.928} C_VEL
LIN {X 0,Y 310.975,Z 614.802,A -85,B 0,C 180,E1 -15562.207,E2 -15562.207} C_VEL
LIN {X 0,Y 310.834,Z 618.783,A -85,B 0,C 180,E1 -15564.181,E2 -15564.181} C_VEL
LIN {X 0,Y 310.8,Z 621.647,A -85,B 0,C 180,E1 -15566.11,E2 -15566.11} C_VEL
LIN {X 0,Y 310.77,Z 623.008,A -85,B 0,C 180,E1 -15567.408,E2 -15567.408} C_VEL
LIN {X 0,Y 310.815,Z 623.972,A -85,B 0,C 180,E1 -15568.704,E2 -15568.704} C_VEL
LIN {X 0,Y 310.856,Z 624.54,A -85,B 0,C 180,E1 -15570,E2 -15570} C_VEL
LIN {X 0,Y 310.774,Z 624.684,A -85,B 0,C 180,E1 -15571.296,E2 -15571.296} C_VEL
LIN {X 0,Y 310.751,Z 623.751,A -85,B 0,C 180,E1 -15573.89,E2 -15573.89} C_VEL
LIN {X 0,Y 310.735,Z 622.236,A -85,B 0,C 180,E1 -15575.637,E2 -15575.637} C_VEL
LIN {X 0,Y 311.009,Z 619.322,A -85,B 0,C 180,E1 -15577.792,E2 -15577.792} C_VEL
LIN {X 0,Y 311.446,Z 615.637,A -85,B 0,C 180,E1 -15579.744,E2 -15579.744} C_VEL
LIN {X 0,Y 312.151,Z 610.857,A -85,B 0,C 180,E1 -15581.691,E2 -15581.691} C_VEL
LIN {X 0,Y 313.548,Z 603.725,A -85,B 0,C 180,E1 -15583.943,E2 -15583.943} C_VEL
LIN {X 0,Y 314.908,Z 596.236,A -85,B 0,C 180,E1 -15585.812,E2 -15585.812} C_VEL
LIN {X 0,Y 316.333,Z 588.13,A -85,B 0,C 180,E1 -15587.452,E2 -15587.452} C_VEL
LIN {X 0,Y 318.081,Z 578.544,A -85,B 0,C 180,E1 -15589.02,E2 -15589.02} C_VEL
LIN {X 0,Y 319.94,Z 567.933,A -85,B 0,C 180,E1 -15590.409,E2 -15590.409} C_VEL
LIN {X 0,Y 321.52,Z 557.704,A -85,B 0,C 180,E1 -15591.477,E2 -15591.477} C_VEL
LIN {X 0,Y 323.146,Z 545.569,A -85,B 0,C 180,E1 -15592.455,E2 -15592.455} C_VEL
LIN {X 0,Y 324.528,Z 532.092,A -85,B 0,C 180,E1 -15593.237,E2 -15593.237} C_VEL
LIN {X 0,Y 325.352,Z 519.604,A -85,B 0,C 180,E1 -15593.723,E2 -15593.723} C_VEL
LIN {X 0,Y 327.067,Z 455.787,A -85,B 0,C 180,E1 -15595.153,E2 -15595.153} C_VEL
LIN {X 0,Y 323.596,Z 434.293,A -85,B 0,C 180,E1 -15596.017,E2 -15596.017} C_VEL
LIN {X 0,Y 319.02,Z 412.353,A -85,B 0,C 180,E1 -15597.034,E2 -15597.034} C_VEL
LIN {X 0,Y 318.801,Z 410.898,A -85,B 0,C 180,E1 -15597.129,E2 -15597.129} C_VEL
LIN {X 0,Y 317.653,Z 404.199,A -85,B 0,C 180,E1 -15599.126,E2 -15599.126} C_VEL
LIN {X 0,Y 315.091,Z 392.772,A -85,B 0,C 180,E1 -15602.743,E2 -15602.743} C_VEL
LIN {X 0,Y 312.507,Z 382.559,A -85,B 0,C 180,E1 -15606.219,E2 -15606.219} C_VEL
LIN {X 0,Y 312.505,Z 382.557,A -85,B 0,C 180,E1 -15609.027,E2 -15609.027} C_VEL
LIN {X 0,Y 312.492,Z 382.556,A -85,B 0,C 180,E1 -15612.43,E2 -15612.43} C_VEL
LIN {X 0,Y 312.534,Z 382.55,A -85,B 0,C 180,E1 -15616.019,E2 -15616.019} C_VEL
LIN {X 0,Y 312.542,Z 382.549,A -85,B 0,C 180,E1 -15619.865,E2 -15619.865} C_VEL
LIN {X 0,Y 312.548,Z 382.547,A -85,B 0,C 180,E1 -15622.618,E2 -15622.618} C_VEL
LIN {X 0,Y 312.514,Z 382.555,A -85,B 0,C 180,E1 -15626.311,E2 -15626.311} C_VEL
LIN {X 0,Y 312.54,Z 382.55,A -85,B 0,C 180,E1 -15630.35,E2 -15630.35} C_VEL
LIN {X 0,Y 312.597,Z 382.526,A -85,B 0,C 180,E1 -15634.064,E2 -15634.064} C_VEL
LIN {X 0,Y 312.581,Z 382.543,A -85,B 0,C 180,E1 -15637.529,E2 -15637.529} C_VEL
LIN {X 0,Y 312.632,Z 382.539,A -85,B 0,C 180,E1 -15641.656,E2 -15641.656} C_VEL
LIN {X 0,Y 312.687,Z 382.531,A -85,B 0,C 180,E1 -15645.686,E2 -15645.686} C_VEL
LIN {X 0,Y 312.697,Z 382.526,A -85,B 0,C 180,E1 -15649.642,E2 -15649.642} C_VEL
LIN {X 0,Y 312.865,Z 382.512,A -85,B 0,C 180,E1 -15652.254,E2 -15652.254} C_VEL
LIN {X 0,Y 312.713,Z 382.525,A -85,B 0,C 180,E1 -15654.843,E2 -15654.843} C_VEL
LIN {X 0,Y 312.986,Z 382.49,A -85,B 0,C 180,E1 -15658.714,E2 -15658.714} C_VEL
LIN {X 0,Y 313.114,Z 382.478,A -85,B 0,C 180,E1 -15660,E2 -15660} C_VEL
LIN {X 0,Y 312.931,Z 382.5,A -85,B 0,C 180,E1 -15662.575,E2 -15662.575} C_VEL
LIN {X 0,Y 312.878,Z 382.511,A -85,B 0,C 180,E1 -15666.635,E2 -15666.635} C_VEL
LIN {X 0,Y 312.761,Z 382.522,A -85,B 0,C 180,E1 -15669.05,E2 -15669.05} C_VEL
LIN {X 0,Y 312.628,Z 382.537,A -85,B 0,C 180,E1 -15672.992,E2 -15672.992} C_VEL
LIN {X 0,Y 312.632,Z 382.54,A -85,B 0,C 180,E1 -15675.65,E2 -15675.65} C_VEL
LIN {X 0,Y 312.625,Z 382.542,A -85,B 0,C 180,E1 -15679.237,E2 -15679.237} C_VEL
LIN {X 0,Y 312.541,Z 382.554,A -85,B 0,C 180,E1 -15682.79,E2 -15682.79} C_VEL
LIN {X 0,Y 312.592,Z 382.524,A -85,B 0,C 180,E1 -15685.934,E2 -15685.934} C_VEL
LIN {X 0,Y 312.541,Z 382.553,A -85,B 0,C 180,E1 -15689.651,E2 -15689.651} C_VEL
LIN {X 0,Y 312.516,Z 382.556,A -85,B 0,C 180,E1 -15693.69,E2 -15693.69} C_VEL
LIN {X 0,Y 312.55,Z 382.552,A -85,B 0,C 180,E1 -15697.382,E2 -15697.382} C_VEL
LIN {X 0,Y 312.524,Z 382.559,A -85,B 0,C 180,E1 -15700.705,E2 -15700.705} C_VEL
LIN {X 0,Y 312.538,Z 382.561,A -85,B 0,C 180,E1 -15704.195,E2 -15704.195} C_VEL
LIN {X 0,Y 312.533,Z 382.563,A -85,B 0,C 180,E1 -15707.91,E2 -15707.91} C_VEL
LIN {X 0,Y 312.579,Z 382.583,A -85,B 0,C 180,E1 -15711.96,E2 -15711.96} C_VEL
LIN {X 0,Y 313.465,Z 386.393,A -85,B 0,C 180,E1 -15713.383,E2 -15713.383} C_VEL
LIN {X 0,Y 322.553,Z 405.21,A -85,B 0,C 180,E1 -15714.839,E2 -15714.839} C_VEL
LIN {X 0,Y 328.046,Z 418.092,A -85,B 0,C 180,E1 -15715.706,E2 -15715.706} C_VEL
LIN {X 0,Y 325.942,Z 492.919,A -85,B 0,C 180,E1 -15717.382,E2 -15717.382} C_VEL
LIN {X 0,Y 325.215,Z 505.446,A -85,B 0,C 180,E1 -15717.895,E2 -15717.895} C_VEL
LIN {X 0,Y 324.163,Z 517.865,A -85,B 0,C 180,E1 -15718.646,E2 -15718.646} C_VEL
LIN {X 0,Y 322.743,Z 529.447,A -85,B 0,C 180,E1 -15719.584,E2 -15719.584} C_VEL
LIN {X 0,Y 321.423,Z 540.4,A -85,B 0,C 180,E1 -15720.764,E2 -15720.764} C_VEL
LIN {X 0,Y 319.704,Z 550.854,A -85,B 0,C 180,E1 -15722.158,E2 -15722.158} C_VEL
LIN {X 0,Y 318.012,Z 560.518,A -85,B 0,C 180,E1 -15723.769,E2 -15723.769} C_VEL
LIN {X 0,Y 316.304,Z 569.428,A -85,B 0,C 180,E1 -15725.643,E2 -15725.643} C_VEL
LIN {X 0,Y 314.69,Z 577.166,A -85,B 0,C 180,E1 -15727.688,E2 -15727.688} C_VEL
LIN {X 0,Y 313.462,Z 583.049,A -85,B 0,C 180,E1 -15729.665,E2 -15729.665} C_VEL
LIN {X 0,Y 312.542,Z 587.636,A -85,B 0,C 180,E1 -15731.651,E2 -15731.651} C_VEL
LIN {X 0,Y 312.015,Z 590.035,A -85,B 0,C 180,E1 -15732.974,E2 -15732.974} C_VEL
LIN {X 0,Y 311.641,Z 591.988,A -85,B 0,C 180,E1 -15734.299,E2 -15734.299} C_VEL
LIN {X 0,Y 311.24,Z 593.981,A -85,B 0,C 180,E1 -15736.163,E2 -15736.163} C_VEL
LIN {X 0,Y 310.885,Z 595.239,A -85,B 0,C 180,E1 -15738.261,E2 -15738.261} C_VEL
LIN {X 0,Y 310.738,Z 595.387,A -85,B 0,C 180,E1 -15740.891,E2 -15740.891} C_VEL
LIN {X 0,Y 310.788,Z 594.826,A -85,B 0,C 180,E1 -15742.202,E2 -15742.202} C_VEL
LIN {X 0,Y 310.95,Z 593.459,A -85,B 0,C 180,E1 -15743.981,E2 -15743.981} C_VEL
LIN {X 0,Y 311.14,Z 589.722,A -85,B 0,C 180,E1 -15746.763,E2 -15746.763} C_VEL
LIN {X 0,Y 311.535,Z 585.887,A -85,B 0,C 180,E1 -15748.707,E2 -15748.707} C_VEL
LIN {X 0,Y 311.995,Z 580.945,A -85,B 0,C 180,E1 -15750.645,E2 -15750.645} C_VEL
LIN {X 0,Y 312.821,Z 574.724,A -85,B 0,C 180,E1 -15752.575,E2 -15752.575} C_VEL
LIN {X 0,Y 313.877,Z 566.941,A -85,B 0,C 180,E1 -15754.495,E2 -15754.495} C_VEL
LIN {X 0,Y 315.007,Z 557.262,A -85,B 0,C 180,E1 -15756.405,E2 -15756.405} C_VEL
LIN {X 0,Y 316.306,Z 547.187,A -85,B 0,C 180,E1 -15757.982,E2 -15757.982} C_VEL
LIN {X 0,Y 317.536,Z 535.798,A -85,B 0,C 180,E1 -15759.394,E2 -15759.394} C_VEL
LIN {X 0,Y 318.498,Z 524.641,A -85,B 0,C 180,E1 -15760.489,E2 -15760.489} C_VEL
LIN {X 0,Y 319.379,Z 513.292,A -85,B 0,C 180,E1 -15761.342,E2 -15761.342} C_VEL
LIN {X 0,Y 320.058,Z 500.359,A -85,B 0,C 180,E1 -15762.04,E2 -15762.04} C_VEL
LIN {X 0,Y 320.494,Z 486.571,A -85,B 0,C 180,E1 -15762.506,E2 -15762.506} C_VEL
LIN {X 0,Y 322.065,Z 412.293,A -85,B 0,C 180,E1 -15764.141,E2 -15764.141} C_VEL
LIN {X 0,Y 320.122,Z 404.75,A -85,B 0,C 180,E1 -15764.446,E2 -15764.446} C_VEL
LIN {X 0,Y 313.195,Z 385.34,A -85,B 0,C 180,E1 -15765.394,E2 -15765.394} C_VEL
LIN {X 0,Y 312.646,Z 382.544,A -85,B 0,C 180,E1 -15766.403,E2 -15766.403} C_VEL
LIN {X 0,Y 312.595,Z 382.546,A -85,B 0,C 180,E1 -15769.708,E2 -15769.708} C_VEL
LIN {X 0,Y 312.549,Z 382.553,A -85,B 0,C 180,E1 -15772.789,E2 -15772.789} C_VEL
LIN {X 0,Y 312.589,Z 382.548,A -85,B 0,C 180,E1 -15776.721,E2 -15776.721} C_VEL
LIN {X 0,Y 312.551,Z 382.549,A -85,B 0,C 180,E1 -15779.649,E2 -15779.649} C_VEL
LIN {X 0,Y 312.521,Z 382.554,A -85,B 0,C 180,E1 -15783.688,E2 -15783.688} C_VEL
LIN {X 0,Y 312.525,Z 382.552,A -85,B 0,C 180,E1 -15787.458,E2 -15787.458} C_VEL
LIN {X 0,Y 312.489,Z 382.557,A -85,B 0,C 180,E1 -15790.708,E2 -15790.708} C_VEL
LIN {X 0,Y 312.486,Z 382.557,A -85,B 0,C 180,E1 -15793.049,E2 -15793.049} C_VEL
LIN {X 0,Y 311.822,Z 382.643,A -85,B 0,C 180,E1 -15794.126,E2 -15794.126} C_VEL
LIN {X 0,Y 308.985,Z 382.994,A -85,B 0,C 180,E1 -15795.878,E2 -15795.878} C_VEL
LIN {X 0,Y 306.583,Z 383.291,A -85,B 0,C 180,E1 -15797.299,E2 -15797.299} C_VEL
LIN {X 0,Y 305.557,Z 383.422,A -85,B 0,C 180,E1 -15798.399,E2 -15798.399} C_VEL
LIN {X 0,Y 305.476,Z 383.427,A -85,B 0,C 180,E1 -15798.771,E2 -15798.771} C_VEL
LIN {X 0,Y 305.518,Z 383.426,A -85,B 0,C 180,E1 -15801.603,E2 -15801.603} C_VEL
LIN {X 0,Y 305.46,Z 383.427,A -85,B 0,C 180,E1 -15804.886,E2 -15804.886} C_VEL
LIN {X 0,Y 305.446,Z 383.439,A -85,B 0,C 180,E1 -15808.355,E2 -15808.355} C_VEL
LIN {X 0,Y 305.509,Z 383.426,A -85,B 0,C 180,E1 -15811.112,E2 -15811.112} C_VEL
LIN {X 0,Y 305.566,Z 383.418,A -85,B 0,C 180,E1 -15814.087,E2 -15814.087} C_VEL
LIN {X 0,Y 305.524,Z 383.428,A -85,B 0,C 180,E1 -15818.404,E2 -15818.404} C_VEL
LIN {X 0,Y 305.586,Z 383.416,A -85,B 0,C 180,E1 -15821.217,E2 -15821.217} C_VEL
LIN {X 0,Y 305.643,Z 383.404,A -85,B 0,C 180,E1 -15825.348,E2 -15825.348} C_VEL
LIN {X 0,Y 305.634,Z 383.411,A -85,B 0,C 180,E1 -15829.399,E2 -15829.399} C_VEL
LIN {X 0,Y 305.806,Z 383.392,A -85,B 0,C 180,E1 -15832.074,E2 -15832.074} C_VEL
LIN {X 0,Y 305.683,Z 383.398,A -85,B 0,C 180,E1 -15834.723,E2 -15834.723} C_VEL
LIN {X 0,Y 305.952,Z 383.372,A -85,B 0,C 180,E1 -15838.683,E2 -15838.683} C_VEL
LIN {X 0,Y 305.952,Z 383.371,A -85,B 0,C 180,E1 -15841.316,E2 -15841.316} C_VEL
LIN {X 0,Y 305.845,Z 383.385,A -85,B 0,C 180,E1 -15846.597,E2 -15846.597} C_VEL
LIN {X 0,Y 305.73,Z 383.398,A -85,B 0,C 180,E1 -15849.26,E2 -15849.26} C_VEL
LIN {X 0,Y 305.584,Z 383.417,A -85,B 0,C 180,E1 -15853.296,E2 -15853.296} C_VEL
LIN {X 0,Y 305.587,Z 383.422,A -85,B 0,C 180,E1 -15856.02,E2 -15856.02} C_VEL
LIN {X 0,Y 305.575,Z 383.418,A -85,B 0,C 180,E1 -15859.447,E2 -15859.447} C_VEL
LIN {X 0,Y 305.484,Z 383.429,A -85,B 0,C 180,E1 -15863.042,E2 -15863.042} C_VEL
LIN {X 0,Y 305.525,Z 383.428,A -85,B 0,C 180,E1 -15866.221,E2 -15866.221} C_VEL
LIN {X 0,Y 305.482,Z 383.43,A -85,B 0,C 180,E1 -15869.047,E2 -15869.047} C_VEL
LIN {X 0,Y 305.437,Z 383.441,A -85,B 0,C 180,E1 -15871.953,E2 -15871.953} C_VEL
LIN {X 0,Y 305.457,Z 383.434,A -85,B 0,C 180,E1 -15875.114,E2 -15875.114} C_VEL
LIN {X 0,Y 305.489,Z 383.43,A -85,B 0,C 180,E1 -15878.54,E2 -15878.54} C_VEL
LIN {X 0,Y 305.505,Z 383.428,A -85,B 0,C 180,E1 -15882.597,E2 -15882.597} C_VEL
LIN {X 0,Y 305.476,Z 383.433,A -85,B 0,C 180,E1 -15886.355,E2 -15886.355} C_VEL
LIN {X 0,Y 305.456,Z 383.439,A -85,B 0,C 180,E1 -15889.893,E2 -15889.893} C_VEL
LIN {X 0,Y 305.497,Z 383.432,A -85,B 0,C 180,E1 -15893.628,E2 -15893.628} C_VEL
LIN {X 0,Y 305.549,Z 383.623,A -85,B 0,C 180,E1 -15897.379,E2 -15897.379} C_VEL
LIN {X 0,Y 308.191,Z 395.991,A -85,B 0,C 180,E1 -15901.069,E2 -15901.069} C_VEL
LIN {X 0,Y 309.632,Z 404.022,A -85,B 0,C 180,E1 -15903.367,E2 -15903.367} C_VEL
LIN {X 0,Y 309.18,Z 409.286,A -85,B 0,C 180,E1 -15904.756,E2 -15904.756} C_VEL
LIN {X 0,Y 308.915,Z 411.349,A -85,B 0,C 180,E1 -15905.293,E2 -15905.293} C_VEL
